# B&R Automation Studio project ProjectOrionBms
Automation Studio 4.12.6.106; technology packages: mapp 5.24.3, mappView 5.24.3

## Configuration Config1

CPU X90CP174.48-00, AutomationRuntime I4.93, Build 4.1.2, Safety 0.0, Vc V4.72.6

### Task classes (Cpu.sw)
```
Cyclic#1 (cycle 1000 us, tolerance 10000 us):
  INS <- INS.INS.prg
Cyclic#2 (cycle 4000 us, tolerance 20000 us):
  AMS_CAN <- AMS_and_Shunt.CAN.AMS_CAN.prg
  INV_CAN <- Inverters.CAN.CAN.prg
Cyclic#3 (cycle 10000 us, tolerance 20000 us):
  INV_CTRL <- Inverters.Control.Control.prg
Cyclic#4 (cycle 20000 us, tolerance 20000 us):
  INV_SM <- Inverters.Inv_statemachine.Inv_statemachine.prg
  SENSORS <- Sensors.Sensors.prg
  ACTUATORS <- Actuators.Output.prg
  DASHBOARD <- Dashboard.Dashboard.prg
  COOLING <- CoolingSystem.COOLING.prg
  file <- File.file.prg
  NewLogging <- Misc.DataLogging.NewLogging.prg
Cyclic#5 (cycle 50000 us, tolerance 50000 us):
  Simulation <- Inverters.Simulation.Simulation.prg [disabled]
  AMS_CTRL <- AMS_and_Shunt.AMS.prg
  SC <- SC.SafetyChain.prg
  SM <- SM.StateMachine.prg
  SENSOR_NET <- SensorNet.globalSensorNet.prg [disabled]
  ALARM_MAN <- Misc.AlarmManagement.AlarmManagement.prg
Cyclic#6 (cycle 100000 us, tolerance 100000 us):
  sampleST <- Misc.DataLogging.sampleST.prg [disabled]
  DATALOG <- Misc.DataLogging.DataLog.prg [disabled]
Binaries: TCData, udbdef, mvLoader, arsvcreg, ashwac, Role, ashwd, arconfig, sysconf, iomap, User, asfw, Config_1, Config, Config_2, Config_3, DataRecord, OpcUaMap, Acp10map, acp10cfg
Libraries: runtime, astime, standard, operator, AsIecCon, AsIODiag, brsystem, asstring, ArCan, brdkSIM, brdkUSB, AsIO, AsBrStr, sys_lib, FileIO, AsUSB, DataObj, brdkSTR, MpAlarmX, MpBase, MpData, NcGlobal, MpRecipe, sduVikings, MTTypes, dvframe, MTFilter, brdkFile, arssl, areventlog
```

### Hardware
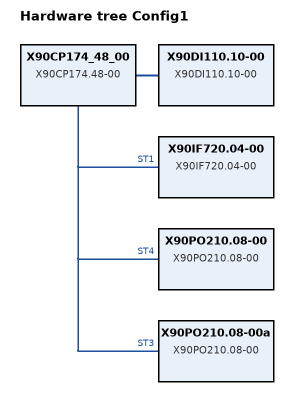
```
X90CP174_48_00 : X90CP174.48-00 v1.5.2.0  [X1 -> X1.SL]
  Module X1 (Type=X1, Virtual=true, Version=1.5.2.0)
    Connection (Connector=SL, TargetModule=X90CP174_48_00, TargetConnector=X1)
    ChannelConfig01 = 42
    DigitalFilterPin01 = 200
    ChannelConfig02 = 42
    DigitalFilterPin02 = 200
    ChannelConfig03 = 42
    DigitalFilterPin03 = 200
    ChannelConfig04 = 42
    DigitalFilterPin04 = 200
    ChannelConfig05 = 42
    DigitalFilterPin05 = 200
    ChannelConfig06 = 42
    DigitalFilterPin06 = 200
    ChannelConfig07 = 42
    DigitalFilterPin07 = 200
    ChannelConfig08 = 42
    DigitalFilterPin08 = 200
    ChannelConfig09 = 80
    ChannelConfig10 = 80
    ChannelConfig11 = 80
    ChannelConfig12 = 81
    ChannelConfig13 = 72
    DigitalFilterPin13 = 200
    ChannelConfig14 = 81
    ChannelConfig16 = 81
    ChannelConfig17 = 80
    ChannelConfig18 = 80
    ChannelConfig19 = 80
    ChannelConfig20 = 80
    ChannelConfig21 = 80
    ChannelConfig22 = 80
    ChannelConfig23 = 80
    IN2_InputFilter_Pin23 = 3
    ChannelConfig24 = 80
    ChannelConfig27 = 1
    ChannelConfig28 = 41
    DigitalFilterPin28 = 200
    ChannelConfig37 = 1
    LoadType37 = 2
    ChannelConfig38 = 1
    LoadType38 = 2
    ChannelConfig39 = 1
    ChannelConfig41 = 1
    LoadType41 = 2
    ChannelConfig42 = 1
    ChannelConfig45 = 1
    LoadType45 = 2
    ChannelConfig46 = 1
    LoadType46 = 2
    core = core1
  Connector IF2:
    ActivateDevice = 1
    Mode = Manual
    InternetAddress = 169.254.143.70
    SubnetMask = 255.255.0.0
    InaNodeNumber = 0
    ActivateSnmp = 2
  Connector IF3:
    DNAConfiguration = manual
    CycleTime = 1000
  ConfigurationID = Project_Config1
  UserPartitionSize = 100
  VolatileGlobalPvSize = 100000000
  IdleTaskClass = 5
  TaskClassIdleTime = 5000
  CyclicTaskClassCount = 6
  Cyclic1Duration = 1000
  Cyclic1Tolerance = 10000
  Cyclic2Duration = 4000
  Cyclic2Tolerance = 20000
  Cyclic3Duration = 10000
  Cyclic3Tolerance = 20000
  Cyclic4Duration = 20000
  Cyclic4Tolerance = 20000
  Cyclic5Duration = 50000
  Cyclic5Tolerance = 50000
  Cyclic6Duration = 100000
  Cyclic6Tolerance = 100000
  Cyclic7Duration = 100000
  Cyclic7Tolerance = 1000000
  Cyclic8Duration = 10000
  Cyclic8Tolerance = 30000000
  FileDevice1
  FileDeviceName1 = C
  FileDevicePath1 = C:/vikings/missions
  FileDevice2
  FileDeviceName2 = plc
  FileDevicePath2 = USER_PATH
  FtpUser1
  FtpUsername1 = viking  // viking
  FtpUserPassword1 = ZkV2vChQEXxJT0bhh2t/N5ZFPz9PChZjZfbJ7hc9Et0=  // viking
  FtpUserSalt1 = vdLLncGP
  FTPAccessRight1 = 0
  FTPdevice1 = ALL
  FtpUser2
  FtpUsername2 = usb  // usb
  FtpUserPassword2 = C1MDbg7H4C+9nkC1XVfE1m47HMH3DB0hBQDZaSBhzO4=  // usb
  FtpUserSalt2 = PgfniPeQ
  FTPAccessRight2 = 0
  FTPdevice2 = USB
  ActivateOpcUa = 1
  OpcUaInformationModels_PV_Version = 1
X90DI110.10-00 : X90DI110.10-00 v1.1.1.0  [ST -> X90CP174_48_00.ST2]
  Mode_DigIn01 = 22k_pnp
  InputFilter01 = 200
  Mode_DigIn02 = 22k_pnp
  InputFilter02 = 200
  Mode_DigIn03 = 22k_pnp
  InputFilter03 = 200
  Mode_DigIn04 = 22k_pnp
  Mode_DigIn05 = 22k_pnp
  Mode_DigIn06 = 22k_pnp
  Mode_DigIn07 = 22k_pnp
  InputFilter07 = 200
  Mode_DigIn08 = 22k_pnp
  Mode_DigIn09 = 22k_pnp
  InputFilter09 = 200
  Mode_DigIn10 = 22k_pnp
  InputFilter10 = 200
X90IF720.04-00 : X90IF720.04-00 v1.0.2.0  [ST -> X90CP174_48_00.ST1]
  Connector IF4:
    Baudrate = 115200
X90PO210.08-00 : X90PO210.08-00 v1.0.2.0  [ST -> X90CP174_48_00.ST4]
X90PO210.08-00a : X90PO210.08-00 v1.0.2.0  [ST -> X90CP174_48_00.ST3]
```

### IoMap.iom - X90CP174_48_00/IoMap.iom
```iecst
VAR_CONFIG
	::gCooling.outputs.do_fan[1] AT %QX."X1".DigitalOutput46;
	::gCooling.inputs.ai_coolingTemp[0] AT %IW."X1".AnalogInput17;
	::gCooling.inputs.ai_coolingTemp[1] AT %IW."X1".AnalogInput19;
	::gCooling.outputs.do_pump[1] AT %QX."X1".DigitalOutput45;
	::gCooling.outputs.do_fan[0] AT %QX."X1".DigitalOutput37;
	::gCooling.outputs.do_pump[0] AT %QX."X1".DigitalOutput38;
	::gSafetyChain.inputs.di_interlockWheelFR_OK AT %IX."X1".DigitalInput05;
	::gSafetyChain.inputs.di_shutdownRight_OK AT %IX."X1".DigitalInput07;
	::gSafetyChain.inputs.di_interlockWheelFL_OK AT %IX."X1".DigitalInput06;
	::gSafetyChain.inputs.di_interlockWheelRR_OK AT %IX."X1".DigitalInput08;
	::gSafetyChain.inputs.di_shutdownLeft_OK AT %IX."X1".DigitalInput01;
	::gSafetyChain.inputs.di_shutdownCockpit_OK AT %IX."X1".DigitalInput02;
	::gSafetyChain.inputs.di_inertiaSwitch_OK AT %IX."X1".DigitalInput03;
	::gSafetyChain.inputs.di_BOTS_OK AT %IX."X1".DigitalInput04;
	::gSafetyChain.inputs.di_TSMS_OK AT %IX."X1".DigitalInput13;
	::gSteeringAngle.inputs.angleSensor AT %IW."X1".AnalogInput20;
	::gTorqueSensor.inputs.torque2 AT %IW."X1".AnalogInput21;
	::gBraking.inputs.ai_brakePressureFront AT %IW."X1".AnalogInput22;
	::gTorqueSensor.inputs.torque1 AT %IW."X1".AnalogInput24;
	::gBraking.inputs.ai_brakePressureRear AT %IW."X1".AnalogInput18;
	::gInverters.inverter[0].inputs.di_deratingActive AT %IX."X90DI110.10-00".DigitalInput06;
	::gInverters.inverter[1].inputs.di_deratingActive AT %IX."X90DI110.10-00".DigitalInput04;
	::gInverters.inverter[2].inputs.di_deratingActive AT %IX."X90DI110.10-00".DigitalInput08;
	::gInverters.inverter[3].inputs.di_deratingActive AT %IX."X90DI110.10-00".DigitalInput05;
	::gInverters.inverter[0].outputs.do_enable AT %QX."X90PO210.08-00a".DigitalOutput01;
	::gInverters.inverter[1].outputs.do_enable AT %QX."X90PO210.08-00a".DigitalOutput07;
	::gInverters.inverter[3].outputs.do_enable AT %QX."X90PO210.08-00a".DigitalOutput06;
	::gInverters.inverter[2].outputs.do_torqueLimitActive AT %QX."X90PO210.08-00a".DigitalOutput02;
	::gInverters.inverter[0].outputs.do_torqueLimitActive AT %QX."X90PO210.08-00a".DigitalOutput03;
	::gInverters.inverter[1].outputs.do_torqueLimitActive AT %QX."X90PO210.08-00a".DigitalOutput08;
	::gInverters.output.do_enableInv34 AT %QX."X90PO210.08-00a".DigitalOutput04;
	::gInverters.inverter[2].outputs.do_enable AT %QX."X90PO210.08-00".DigitalOutput03;
	::gInverters.inverter[3].outputs.do_torqueLimitActive AT %QX."X90PO210.08-00".DigitalOutput02;
	::gInverters.output.do_enableInv12 AT %QX."X90PO210.08-00".DigitalOutput05;
	::gSafetyChain.inputs.di_TS_Container AT %IX."X90DI110.10-00".DigitalInput07;
	::gSafetyChain.inputs.di_interlockWheelRL_OK AT %IX."X90DI110.10-00".DigitalInput10;
	::gSafetyChain.inputs.di_supply AT %IX."X90DI110.10-00".DigitalInput09;
	::gSafetyChain.inputs.di_BSPD_OK AT %IX."X90DI110.10-00".DigitalInput03;
	::gSafetyChain.inputs.di_interlockHVD_OK AT %IX."X90DI110.10-00".DigitalInput01;
	::gSafetyChain.inputs.di_interlockTSMP_OK AT %IX."X90DI110.10-00".DigitalInput02;
	::gRTDS.outputs.do_RTDS AT %QX."X1".DigitalOutput41;
	::gBraking.outputs.do_brakeLight AT %QX."X1".DigitalOutput42;
	gRTDS.inputs.im_RTDS_Current AT %IW."X1".Current41;
	::gCooling.inputs.im_pumpCurrent[1] AT %IW."X1".Current45;
	::gCooling.inputs.im_pumpCurrent[0] AT %IW."X1".Current38;
	::gInverters.output.do_powerInv12 AT %QX."X1".DigitalOutput39;
	::gInverters.output.do_powerInv34 AT %QX."X1".DigitalOutput27;
	::gLowVoltageBattery.inputs.ai_voltage AT %IW."X1".AnalogInput12;
	::gLowVoltageBattery.inputs.ai_current AT %IW."X1".AnalogInput23;
	::gSafetyChain.inputs.di_interlockMotorRL_OK AT %IX."X1".DigitalInput28;
	::SENSORS:suspension.input.linearPosSensor[2] AT %IW."X1".AnalogInput16;
	::SENSORS:suspension.input.linearPosSensor[0] AT %IW."X1".AnalogInput14;
	::SENSORS:accelerometer.input.z_direction AT %IW."X1".AnalogInput09;
	::SENSORS:accelerometer.input.y_direction AT %IW."X1".AnalogInput10;
	::SENSORS:accelerometer.input.x_direction AT %IW."X1".AnalogInput11;
END_VAR
```

### Config_2.mpdatarecorder - X90CP174_48_00/mappServices/Config_2.mpdatarecorder
```
Element gDataRecorder (Type=mpdatarecorder)
  DataRecorder:
    MaxFileSize = 32000
    SaveInterval = 5000
```

### DataRecord.mpdatarecorder - X90CP174_48_00/mappServices/DataRecord.mpdatarecorder
```
Element gDataRecorderNew (Type=mpdatarecorder)
  DataRecorder:
    MaxNumberOfFiles = 4
    MaxFileSize = 32000
    DecimalDigits = 3
    SaveInterval = 2000
    FileNamePattern = Datalog_%H_%M_%S.csv
    TimeStampPattern = %H:%M:%S:%L
```

## Logical view

Binary libraries used (declarations not repeated): operator, runtime, astime, AsIecCon, standard, AsIODiag, brsystem, asstring, ArCan, brdkSIM, AsIO, AsBrStr, sys_lib, FileIO, AsUSB, DataObj, brdkSTR, NcGlobal, MTTypes 1.03.4, dvframe, MTFilter, MpAlarmX 5.24.3, MpBase, MpRecipe 5.24.3, MpData 5.24.3

- AS4_HW_X90PO210.08-00.exe (binary file, 1100199 bytes)
### Global.var - Global variables
```iecst
VAR
	gIsSimulation : BOOL;
END_VAR
```

### Package Logical/Libraries - Global libraries

### Library Logical/Libraries/brdkUSB (ANSIC, version 1.00.3)
Depends on: AsUSB, FileIO

#### brdkUSBConnect.c
```c
#include <bur/plctypes.h>
#include <string.h>
#ifdef __cplusplus
	extern "C"
	{
#endif

	#include "brdkUSB.h"

#ifdef __cplusplus
	};
#endif

#define true 1
#define false 0

/* Converts an UDINT into a STRING type */
static unsigned char brdkUSBuditoa(unsigned long Value, char* pString) {
	int i, j=0;
	pString[0] = 0;
	if (Value > 0) {
		while (Value > 0) {
			j++;
			for(i=j; i > 0 ; i--) {
				pString[i] =pString[i-1];
			}
			pString[0] = (Value % 10) + 48;			/* ASCII 48-57 = 0..9 */
			Value = (Value / 10);
		}
	}
	else {
		pString[0] = 48;								/* adds just a zero char  */
		pString[1] = 0;								/* ends the string  */
		j = 1;
	}
	return j;
}

void brdkUSBConnect(struct brdkUSBConnect* inst) {
	brdk_usb_connect_internal_typ* this = &inst->internal;
	int i,n,idx;
	char tmp[2];

	/* get list of all connected usb nodes */
	this->UsbNodeListGet_0.enable 					= true;
	this->UsbNodeListGet_0.pBuffer					= (UDINT)&this->nodeIdBuffer;
	this->UsbNodeListGet_0.bufferSize 				= sizeof(this->nodeIdBuffer);
	this->UsbNodeListGet_0.filterInterfaceClass 	= asusb_CLASS_MASS_STORAGE;
	this->UsbNodeListGet_0.filterInterfaceSubClass 	= 0;
	UsbNodeListGet(&this->UsbNodeListGet_0);
	if(this->UsbNodeListGet_0.status == ERR_OK || (this->UsbNodeListGet_0.status == asusbERR_USB_NOTFOUND && this->UsbNodeListGet_0.listNodes == 0)) {

		if(this->oldCnt != this->UsbNodeListGet_0.listNodes && this->UsbNodeListGet_0.listNodes > 0) {

			/* go through all list nodes and check if they have been added to the system */
			for (n = 0; n < this->UsbNodeListGet_0.listNodes; n++) {
				idx = -1;
				for (i = 0; i <= BRDK_USB_MAX_DEVICES; i++) {
					if (this->node[i].UsbNodeGet_0.nodeId == this->nodeIdBuffer[n]) {
						idx = this->nodeIdBuffer[n];
						break;
					}
				}
				if (idx == -1) {	/* device not found/added */
					for (i = 0; i <= BRDK_USB_MAX_DEVICES; i++) {
						if (this->node[i].UsbNodeGet_0.nodeId == 0) {
							this->node[i].UsbNodeGet_0.nodeId = this->nodeIdBuffer[n];
							break;
						}
					}
				}
			}
		}
		this->oldCnt = this->UsbNodeListGet_0.listNodes;
	}
	else if(inst->simulateMount && !this->simulationMountActivated) {
	/* find an avaible node index */
		for(i=0; i<= BRDK_USB_MAX_DEVICES; i++) {
			if(this->node[i].UsbNodeGet_0.nodeId == 0) {
				this->node[i].UsbNodeGet_0.nodeId = 4294967295LL;
				this->simulationMountActivated = true;
				break;
			}
		}
	}

	/* state machine for all usb nodes */
	for(i=0; i<= BRDK_USB_MAX_DEVICES; i++) {

		switch(this->node[i].state) {

			case 0: /* wait for id */
				if(this->node[i].UsbNodeGet_0.nodeId != 0) {
					this->node[i].UsbNodeGet_0.enable 		= (this->node[i].UsbNodeGet_0.nodeId < 4294967294LL);
					this->node[i].UsbNodeGet_0.pBuffer 		= (UDINT)&this->node[i].infoBuffer;
					this->node[i].UsbNodeGet_0.bufferSize 	= sizeof(usbNode_typ);
					UsbNodeGet(&this->node[i].UsbNodeGet_0);
					this->node[i].state 					= 10;
				}
				break;

			case 10:	/* get usb node info (interface name) */
				UsbNodeGet(&this->node[i].UsbNodeGet_0);
				switch(this->node[i].UsbNodeGet_0.status) {

					case ERR_OK:
						/* filter B&R technology guard from list */
						if(this->node[i].infoBuffer.vendorId == 1615 && this->node[i].infoBuffer.productId == 1001) this->node[i].state = 70;
						else {
							strcpy(this->node[i].device,"USB");
							brdkUSBuditoa(i,tmp);
							strcat(this->node[i].device,tmp);
							this->node[i].DevLink_0.pDevice = (UDINT)&this->node[i].device;
							strcpy(this->node[i].param, "/DEVICE=");
							strcat(this->node[i].param, this->node[i].infoBuffer.ifName);
							this->node[i].DevLink_0.pParam = (UDINT)&this->node[i].param;
							this->node[i].DevLink_0.enable = true;
							this->node[i].state = 20;
						}
						break;

					case asusbERR_USB_NOTFOUND:
						this->node[i].UsbNodeGet_0.nodeId = 0;
						memset(&this->node[i].infoBuffer,0,sizeof(usbNode_typ));
						this->node[i].state = 0;
						break;

					case ERR_FUB_ENABLE_FALSE:
						strcpy(this->node[i].device,"USB");
						brdkUSBuditoa(i,tmp);
						strcat(this->node[i].device,tmp);
						this->node[i].DevLink_0.pDevice = (UDINT)&this->node[i].device;
						strcpy(this->node[i].param, "/DEVICE=C:\\USB");
						this->node[i].DevLink_0.pParam = (UDINT)&this->node[i].param;
						this->node[i].DevLink_0.enable = true;
						this->node[i].state = 20;
						break;

				}
				break;

			case 20:	/* create device link */
				DevLink(&this->node[i].DevLink_0);
				switch(this->node[i].DevLink_0.status) {

					case ERR_OK:
						strcpy(inst->node[i].device,this->node[i].device);
						this->node[i].state = 40;
						break;

					case fiERR_DEVICE_ALREADY_EXIST:
						this->node[i].DevUnlink_0.enable 	= 1;
						this->node[i].DevUnlink_0.handle 	= this->node[i].DevLink_0.handle;
						this->node[i].state 				= 30;
						break;
				}
				break;

			case 30:	/* unlink device link */
				DevUnlink(&this->node[i].DevUnlink_0);
				switch(this->node[i].DevUnlink_0.status ) {

					case ERR_OK: case fiERR_DEVICE_INVALID_HANDLE:
						this->node[i].DevUnlink_0.enable 	= 0;
						DevUnlink(&this->node[i].DevUnlink_0);
						this->node[i].DevLink_0.enable 		= 0;
						DevLink(&this->node[i].DevLink_0);
						this->node[i].DevLink_0.enable 		= 1;
						this->node[i].devLinkFailCnt++;
						brdkUSBuditoa(this->node[i].devLinkFailCnt,tmp);
						strcat(this->node[i].device,tmp);
						this->node[i].DevLink_0.pDevice 	= (UDINT)&this->node[i].device;
						this->node[i].state					= 20;
						break;

				}
				break;

			case 40:	/* usb node ready - monitor node */
				UsbNodeGet(&this->node[i].UsbNodeGet_0);
				switch(this->node[i].UsbNodeGet_0.status) {

					case ERR_OK:
						if(inst->updateMemInfo || inst->node[i].totalMemory == 0) {
							this->node[i].DevMemInfo_0.enable = true;
							this->node[i].DevMemInfo_0.pDevice = this->node[i].DevLink_0.pDevice;
							this->node[i].state = 50;
						}
						break;

					case asusbERR_USB_NOTFOUND:
						strcpy(inst->node[i].device,"");
						this->node[i].DevUnlink_0.enable 	= true;
						this->node[i].DevUnlink_0.handle 	= this->node[i].DevLink_0.handle;
						this->node[i].state = 60;
						break;

					case ERR_FUB_ENABLE_FALSE:
						if(!inst->simulateMount && this->simulationMountActivated) {
							strcpy(inst->node[i].device,"");
							this->node[i].DevUnlink_0.enable 	= true;
							this->node[i].DevUnlink_0.handle 	= this->node[i].DevLink_0.handle;
							this->simulationMountActivated 		= false;
							this->node[i].state = 60;
						}
						break;

				}
				break;

			case 50:	/* read meminfo */
				DevMemInfo(&this->node[i].DevMemInfo_0);
				switch(this->node[i].DevMemInfo_0.status) {

					case ERR_OK:
						inst->node[i].freeMemory 	= this->node[i].DevMemInfo_0.freemem/1048576;	/* output must be in mb */
						inst->node[i].totalMemory 	= this->node[i].DevMemInfo_0.memsize/1048576;	/* output must be in mb */
						this->node[i].state 		= 40;
						break;

					case fiERR_DETMEMINFO: case fiERR_DEVICE_MANAGER:
						inst->node[i].freeMemory 	= -1;	/* output must be in mb */
						inst->node[i].totalMemory 	= -1;	/* output must be in mb */
						this->node[i].state 		= 40;
						break;

					case ERR_FUB_BUSY: break;
					default: this->node[i].state = 40; break;
				}
				break;

			case 60:	/* unlink device */
				DevUnlink(&this->node[i].DevUnlink_0);
				switch(this->node[i].DevUnlink_0.status ) {

					case ERR_OK: case fiERR_DEVICE_INVALID_HANDLE:
						this->node[i].DevUnlink_0.enable 	= false;
						DevUnlink(&this->node[i].DevUnlink_0);
						this->node[i].DevLink_0.enable 		= false;
						DevLink(&this->node[i].DevLink_0);
						this->node[i].UsbNodeGet_0.nodeId = 0;
						memset(&this->node[i].infoBuffer,0,sizeof(usbNode_typ));
						inst->node[i].freeMemory 	= 0;
						inst->node[i].totalMemory 	= 0;
						this->node[i].state = 0;
						break;

				}
				break;

			case 70:	/* B&R technology guard state */
				UsbNodeGet(&this->node[i].UsbNodeGet_0);
				switch(this->node[i].UsbNodeGet_0.status) {

					case ERR_OK: break;

					case asusbERR_USB_NOTFOUND:
						this->node[i].UsbNodeGet_0.nodeId = 0;
						memset(&this->node[i].infoBuffer,0,sizeof(usbNode_typ));
						this->node[i].state = 0;
						break;

				}
				break;

			case 1000:	/* simulate usb device */

				break;

		}
	}

	/* output status */
	for(i=0; i<= BRDK_USB_MAX_DEVICES; i++) {
		if(inst->node[i].device[0] != 0) {
			inst->status = BRDK_USB_STATUS_FB_READY;
			break;
		}
		else inst->status = BRDK_USB_STATUS_NO_USB_DEV_FOUND;
	}

	inst->updateMemInfo = 0;	/* reset update command */

}
```

### Library Logical/Libraries/sduVikings (IEC)

#### launchProfile.st
```iecst
FUNCTION_BLOCK launchProfile
	IF enable THEN

	ELSE
		FOR i := 0 TO 3 DO
			derating_output[i] := 1;
		END_FOR;
	END_IF;

END_FUNCTION_BLOCK
```

#### regenerativeBraking.st
```iecst
(* TODO: Add your comment here *)
FUNCTION_BLOCK regenerativeBraking
	IF NOT enable OR vehicle_lon_velocity < 5 OR torque_pedal > 0 THEN
		// Regenerative braking should be disabled if:
		//	 - Function block is not enabled
		// 	 - The vehicle velocity is below 5km/h
		//   - The torque pedal is pressed
		FOR i := 0 TO 3 DO
			negTrqLimSetpoint[i] := 0;
		END_FOR;
	ELSE
		// Regenerative braking is allowed
		IF brake_pressure = 0 THEN
			// Idle braking
			FOR i := 0 TO 3 DO
				negTrqLimSetpoint[i] := IDLE_MOTOR_TORQUE;
			END_FOR;
		ELSE
			// Control braking from brake pressure
			FOR i := 0 TO 3 DO
				// Calculate regen braking setpoint
				// Current algorithm is linear with the brake pressure offset by the idle motor torque
				// setpoint = idle_torque + gain * brake_pressure
				// The setpoint is then limited to within [0,1]
				negTrqLimSetpoint[i] := LIMIT(0, IDLE_MOTOR_TORQUE + REGEN_BRAKING_GAIN * brake_pressure, 1);
			END_FOR;
			// The setpoint can then be changed with the negative torque transfer from the TV algorithm
			// and limited to within [0,1]
			// Left, [0]&[2]
			negTrqLimSetpoint[0] := LIMIT(0, negTrqLimSetpoint[0] + negative_torque_transfer, 1);
			negTrqLimSetpoint[2] := LIMIT(0, negTrqLimSetpoint[2] + negative_torque_transfer, 1);
			// Right, [1]&[3]
			negTrqLimSetpoint[1] := LIMIT(0, negTrqLimSetpoint[1] - negative_torque_transfer, 1);
			negTrqLimSetpoint[3] := LIMIT(0, negTrqLimSetpoint[3] - negative_torque_transfer, 1);
		END_IF;
	END_IF;

	FOR i := 0 TO 3 DO
		negative_torque_limit[i] := 0;
		positive_torque_limit[i] := 1;
	END_FOR;
END_FUNCTION_BLOCK
```

#### torqueLimiter.st
```iecst
FUNCTION_BLOCK torqueLimiter

	IF enable THEN
		FOR i := 0 TO 3 DO
			derating_output[i] := max_torque/100.00;
		END_FOR;
	ELSE
		FOR i := 0 TO 3 DO
			derating_output[i] := 1;
		END_FOR;
	END_IF;

END_FUNCTION_BLOCK
```

#### tractionControl.st
```iecst
FUNCTION_BLOCK tractionControl
	IF enable THEN

	ELSE
		FOR i := 0 TO 3 DO
			derating_output[i] := 1;
		END_FOR;
	END_IF;

END_FUNCTION_BLOCK
```

### Library Logical/Libraries/brdkFile (ANSIC, version 2.00.0) - File handling library. Makes it easy to handle file devices and to do file handling.
Depends on: AsIODiag, AsUSB, FileIO, brdkSTR

#### brdkFile.typ - Data types
```iecst
TYPE
	brdk_file_dev_handler_int_typ : 	STRUCT  (*Internal variables.*)
		fileState : UINT; (*State of the file device handler.*)
		driveState : UINT; (*State of the drive handler.*)
		DevLink_0 : DevLink; (*Device link.*)
		DevUnlink_0 : DevUnlink; (*Device unlink.*)
		DirInfo_0 : DirInfo; (*Directory create.*)
		driveInternal : STRING[10]; (*Internal drive.*)
		drive : STRING[10]; (*Drive.*)
		deviceParam : STRING[BRDK_FILE_MAX_PATH_LEN]; (*Device parameter string.*)
		fileIdx : DINT; (*File index.*)
		activeHandles : ARRAY[0..BRDK_FILE_MAX_FILES_DEVICES_]OF UDINT; (*Active handles.*)
		internalRootHandle : UDINT; (*Internal drive.*)
		driveReady : BOOL; (*Drive ready to use.*)
		oldUseUSB : BOOL; (*Holds the old command.*)
		oldFileDeviceUseUSB : ARRAY[0..BRDK_FILE_MAX_FILES_DEVICES]OF BOOL; (*Holds the old command for each file device.*)
		usbOK : BOOL; (*USB drive present and ready to use.*)
		brdkFileCreateSubFolders_0 : brdkFileCreateSubFolders; (*Create sub folders.*)
		UsbNodeListGet_0 : UsbNodeListGet; (*Get list of USB nodes.*)
		UsbNodeGet_0 : UsbNodeGet; (*Get USB node.*)
		nodeId : ARRAY[0..BRDK_FILE_MAX_USB_NODES]OF UDINT; (*Node id buffer list.*)
		nodeIdx : USINT; (*Node id index.*)
		usbNode : usbNode_typ; (*Node info.*)
		oldUSBok : BOOL; (*Holds the old status.*)
		oldNodeId : UDINT; (*Holds the old node id.*)
		availableDeviceIndex : DINT; (*Last array index used in the available devices array*)
		availableUsbIndex : DINT; (*Last array index used in the available usb devices array*)
	END_STRUCT;
	brdk_file_dev_handler_sim_typ : 	STRUCT  (*Simulation options.*)
		pcRootFolder : STRING[BRDK_FILE_MAX_PATH_LEN] := 'plcRoot'; (*Path on the PC that will simulate the root of the controller. Default plcRoot -> C:\plcRoot\*)
		pcUSBDrive : brdk_file_drive_typ := D_DRIVE; (*Drive letter of the PC's USB. Default D:\.*)
		pcHDDrive : brdk_file_drive_typ := C_DRIVE; (*Drive letter of the PC's HD. Default C:\.*)
	END_STRUCT;
	brdk_file_dev_handler_setup_typ : 	STRUCT  (*Setup options.*)
		plcDrive : brdk_file_drive_typ := C_DRIVE; (*Drive letter of the controller flash. Default C:\.*)
		usbOverrule : BOOL := FALSE; (*Inserted USB stick will overrule internal flash if the USB stick is present.*)
		fileDevices : ARRAY[0..BRDK_FILE_MAX_FILES_DEVICES]OF brdk_file_file_devices_typ; (*File devices.*)
	END_STRUCT;
	brdk_file_drive_typ :
		( (*Drive selection. Default C:\.*)
		C_DRIVE := 0, (*C:\*)
		D_DRIVE := 1, (*D:\*)
		E_DRIVE := 2, (*E:\*)
		F_DRIVE := 3, (*F:\*)
		G_DRIVE := 4 (*G:\*)
		) := C_DRIVE;
	brdk_file_file_devices_typ : 	STRUCT  (*File devices setup.*)
		name : STRING[BRFK_FILE_MAX_FILE_DEVICE_LEN]; (*Name of the file device to be used as input for file functions.*)
		path : STRING[BRDK_FILE_MAX_PATH_LEN]; (*Folder path for the file device. Only the folders must be entered the drive is setup in the setup options. E.g. config.*)
		useUSB : BOOL := TRUE; (*Enable or disable that device can use a USB device. (True = Use USB if possible, False = Never use USB)*)
	END_STRUCT;
	brdk_file_create_subfold_int_typ : 	STRUCT  (*Internal variables.*)
		state : DINT; (*State of the function block.*)
		DirCreate_0 : DirCreate; (*Directory create.*)
		tmpPath : STRING[BRDK_FILE_MAX_PATH_LEN]; (*Temp path string.*)
		pathPos : DINT; (*Path position.*)
		tmpPathPos : DINT; (*Tmp path position.*)
		tmpLen : DINT; (*Temp length.*)
	END_STRUCT;
	brdk_file_read_internal_typ : 	STRUCT  (*Internal variables.*)
		state : DINT; (*State of the function block.*)
		FileOpen_0 : FileOpen; (*File open.*)
		FileClose_0 : FileClose; (*File close.*)
		FileRead_0 : FileRead; (*File read.*)
		offset : UDINT; (*Read offset.*)
	END_STRUCT;
	brdk_file_write_internal_typ : 	STRUCT  (*Internal variables.*)
		state : DINT; (*State of the function block.*)
		FileOpen_0 : FileOpen; (*File open.*)
		FileCreate_0 : FileCreate; (*File create.*)
		FileClose_0 : FileClose; (*File close.*)
		FileDelete_0 : FileDelete; (*File delete.*)
		FileWrite_0 : FileWrite; (*File write.*)
	END_STRUCT;
END_TYPE
```

#### brdkFile.var - Constants
```iecst
VAR CONSTANT
	BRDK_FILE_MAX_USB_NODES : USINT := 5; (*Maximum number of connected USB nodes. (5 means 6)*)
	BRDK_FILE_MAX_FILES_DEVICES_ : USINT := 10; (*Maximum numbers of file devices. (10 means 10)*)
	BRDK_FILE_MAX_FILES_DEVICES : USINT := 9; (*Maximum numbers of file devices. (9 means 10)*)
	BRDK_FILE_MAX_PATH_LEN : UINT := 200; (*Maximum length of a path.*)
	BRFK_FILE_MAX_FILE_DEVICE_LEN : UINT := 50; (*Maximum length of file device names.*)
END_VAR
```

#### brdkFile.fun - Functions and function blocks
```iecst
FUNCTION_BLOCK brdkFileDeviceHandler (*Easy file device handler. This function block makes file device handling easy. The idea of the function block is that you only need to create one file device name that can be used for both internal and usb flash.*) (*$GROUP=User,$CAT=User,$GROUPICON=User.png,$CATICON=User.png*)
	VAR_INPUT
		enable : BOOL := FALSE; (*Enables the function block.*)
		setup : brdk_file_dev_handler_setup_typ; (*Setup options.*)
		simulation : brdk_file_dev_handler_sim_typ; (*Simulation options.*)
		useUSB : BOOL := FALSE; (*Stores on the USB if it is possible. Can be auto selected in the setup options.*)
	END_VAR
	VAR_OUTPUT
		availableUSB : ARRAY[0..BRDK_FILE_MAX_FILES_DEVICES] OF STRING[BRFK_FILE_MAX_FILE_DEVICE_LEN]; (*List of available USB devices.*)
		availableDevices : ARRAY[0..BRDK_FILE_MAX_FILES_DEVICES] OF STRING[BRFK_FILE_MAX_FILE_DEVICE_LEN]; (*List of available PLC devices.*)
		ready : BOOL := FALSE; (*Means that all file devices have been created and are ready to use.*)
		description : STRING[200] := ''; (*Status description.*)
		status : UINT := 0; (*Status of FileIO function blocks.*)
	END_VAR
	VAR
		internal : brdk_file_dev_handler_int_typ; (*Internal variables.*)
	END_VAR
END_FUNCTION_BLOCK

FUNCTION_BLOCK brdkFileCreateSubFolders (*Creates folders based on a path string.*) (*$GROUP=User,$CAT=User,$GROUPICON=User.png,$CATICON=User.png*)
	VAR_INPUT
		enable : BOOL := FALSE; (*Enables the function block.*)
		path : STRING[BRDK_FILE_MAX_PATH_LEN] := ''; (*Path of folder to be created. Use \ to seperate folders.*)
		fileDevice : STRING[BRFK_FILE_MAX_FILE_DEVICE_LEN] := ''; (*File device name.*)
	END_VAR
	VAR_OUTPUT
		description : STRING[200] := ''; (*Status description.*)
		done : BOOL := FALSE; (*Function block done.*)
		status : UINT := 0; (*Status of DirCreate function block.*)
	END_VAR
	VAR
		internal : brdk_file_create_subfold_int_typ; (*Internal variables.*)
	END_VAR
END_FUNCTION_BLOCK

FUNCTION_BLOCK brdkFileWrite (*Write data to a file.*) (*$GROUP=User,$CAT=User,$GROUPICON=User.png,$CATICON=User.png*)
	VAR_INPUT
		enable : BOOL := FALSE; (*Enables the function block.*)
		pFileDevice : UDINT := 0; (*String pointer to file device.*)
		pFileName : UDINT := 0; (*String pointer to file name.If the file does not exist it will be created.*)
		pData : UDINT := 0; (*Pointer to the data that must be written to the file.*)
		dataLength : UDINT := 0; (*Length of the data that must be written. If 0 is specified \0 will end the data.*)
		overwrite : BOOL := FALSE; (*Overwrite existing file. If not set the data will be appended to existing file.*)
	END_VAR
	VAR_OUTPUT
		status : UINT := 0; (*Status of the function block.*)
	END_VAR
	VAR
		internal : brdk_file_write_internal_typ; (*Internal variables.*)
	END_VAR
END_FUNCTION_BLOCK

FUNCTION_BLOCK brdkFileRead (*Read data from a file.*) (*$GROUP=User,$CAT=User,$GROUPICON=User.png,$CATICON=User.png*)
	VAR_INPUT
		enable : BOOL := FALSE; (*Enables the function block.*)
		pFileDevice : UDINT := 0; (*String pointer to file device.*)
		pFileName : UDINT := 0; (*String pointer to file name.*)
		pData : UDINT := 0; (*Pointer to the data where the data is read to.*)
		dataLength : UDINT := 0; (*Length of the read data buffer.*)
	END_VAR
	VAR_OUTPUT
		status : UINT := 0; (*Status of the function block.*)
		readLength : UDINT := 0; (*Length of the read data.*)
	END_VAR
	VAR
		internal : brdk_file_read_internal_typ; (*Internal variables.*)
	END_VAR
END_FUNCTION_BLOCK
```

#### brdkFileDeviceHandler.c - Easy file device handler.
```c
#include <brdkFile_func.h>

#define BR_TG_VENDOR_ID 1615
#define BR_TG_PRODUCT_ID 1001

void brdkFileDeviceHandler(struct brdkFileDeviceHandler* inst) {
	brdk_file_dev_handler_int_typ* this 	= (brdk_file_dev_handler_int_typ*)&inst->internal;		/* pointer to the internal structure */
	brdk_file_dev_handler_setup_typ* setup 	= (brdk_file_dev_handler_setup_typ*)&inst->setup;		/* pointer to the setup structure */
	brdk_file_dev_handler_sim_typ* sim 		= (brdk_file_dev_handler_sim_typ*)&inst->simulation;	/* pointer to the simulation structure */
	char tmpStr[200];

	if(inst->enable) {

		/* check whether the controller is beeing simulated and watch the usb status */
		if(!DiagCpuIsSimulated()) {
			if(!this->UsbNodeGet_0.enable) this->UsbNodeListGet_0.enable = true;
			this->UsbNodeListGet_0.pBuffer					= (unsigned long)&this->nodeId;
			this->UsbNodeListGet_0.bufferSize 				= sizeof(this->nodeId);
			this->UsbNodeListGet_0.filterInterfaceClass 	= asusb_CLASS_MASS_STORAGE;
			this->UsbNodeListGet_0.filterInterfaceSubClass 	= asusb_SUBCLASS_SCSI_COMMAND_SET;
			UsbNodeListGet(&this->UsbNodeListGet_0);
			if(this->UsbNodeListGet_0.status == asusbERR_USB_NOTFOUND) {
				this->nodeIdx 	= 0;
				this->usbOK 	= false;
			}

			this->UsbNodeGet_0.enable 		= true;
			this->UsbNodeGet_0.nodeId 		= this->nodeId[this->nodeIdx];
			this->UsbNodeGet_0.pBuffer 		= (unsigned long)&this->usbNode;
			this->UsbNodeGet_0.bufferSize 	= sizeof(this->usbNode);
			UsbNodeGet(&this->UsbNodeGet_0);
			if(this->UsbNodeGet_0.status == ERR_OK) {
				if(this->usbNode.vendorId == BR_TG_VENDOR_ID && this->usbNode.productId == BR_TG_PRODUCT_ID) {
					this->UsbNodeGet_0.enable = false;
					UsbNodeGet(&this->UsbNodeGet_0);
					this->nodeIdx++;
				}
				else this->usbOK = true;
			}
			else if(this->UsbNodeGet_0.status == asusbERR_USB_NOTFOUND) {
				this->UsbNodeListGet_0.enable = true;
				this->nodeIdx = 0;
				this->usbOK = false;
			}
			if(this->oldNodeId != this->UsbNodeGet_0.nodeId) this->usbOK = false;
			this->oldNodeId = this->UsbNodeGet_0.nodeId;
		}
		else {
			/* look for USB root folder */
			if(this->DirInfo_0.pDevice != 0) {
				this->DirInfo_0.enable 	= true;
				this->DirInfo_0.pPath 	= (unsigned long)"";
				DirInfo(&this->DirInfo_0);
				switch(this->DirInfo_0.status) {
					case 0: this->usbOK = true; break;
					case 20723: this->usbOK = false; break;
					default: break;
				}
			}
		}
		if(setup->usbOverrule) inst->useUSB = this->usbOK;	/* USB stick will overrule */
	}
	else {
		this->usbOK 					= false;
		this->nodeIdx 					= 0;
		this->DirInfo_0.enable 			= false;
		DirInfo(&this->DirInfo_0);
		this->UsbNodeGet_0.enable 		= false;
		UsbNodeGet(&this->UsbNodeGet_0);
		this->UsbNodeListGet_0.enable 	= false;
		UsbNodeListGet(&this->UsbNodeListGet_0);
	}

	/* drive handler */
	switch(this->driveState) {

		case 0:
			if(inst->enable) {
				if(!DiagCpuIsSimulated()) {										// If the plc is not simulated
					if((inst->useUSB && this->usbOK) || !inst->useUSB) {
						this->driveReady = true;
						if(!inst->useUSB)getDrive(setup->plcDrive,this->drive);
						else brdkStrCpy((unsigned long)this->drive,(unsigned long)this->usbNode.ifName);
						getDrive(setup->plcDrive,this->driveInternal);
						this->driveState = 499;
					}
				}
				else {															// If the plc is simulated
					this->DevLink_0.enable 	= true;
					this->DevLink_0.pDevice = (unsigned long)"INTUSB";
					this->DevLink_0.pParam 	= buildParameterString(getDrive(sim->pcUSBDrive,this->drive),(char*)&"",(char*)&this->deviceParam);
					brdkStrCpy((unsigned long)this->driveInternal, (unsigned long) this->drive);
					this->driveState 		= 100;
				}
			}
			break;

		case 100:	/* create a file device for finding an attached usb flash */
			DevLink(&this->DevLink_0);
			if(this->DevLink_0.status != ERR_FUB_BUSY) {
				if(this->DevLink_0.status == ERR_OK || this->DevLink_0.status == fiERR_DEVICE_ALREADY_EXIST) {
					this->DirInfo_0.pDevice = this->DevLink_0.pDevice;
					this->DevLink_0.enable 	= false;
					DevLink(&this->DevLink_0);
					this->driveState 		= 110;
				}
				else {
					inst->status = this->DevLink_0.status;
					this->DevLink_0.enable 	= false;
					DevLink(&this->DevLink_0);
					brdkStrCpy((unsigned long)inst->description,(unsigned long)"error calling DevLink. Flip enable to reset fb.");
					this->driveState = 900;
				}
			}
			break;

		case 110:	/* wait for DirInfo to have been call once. Fb is call above */
			switch(this->DirInfo_0.status) {

				case 0: case 20723:
					if(!inst->useUSB) {
						getDrive(sim->pcHDDrive,this->drive);
						brdkStrCat((unsigned long)this->drive,(unsigned long)sim->pcRootFolder);
					}
					else getDrive(sim->pcUSBDrive,this->drive);
					getDrive(sim->pcHDDrive,this->driveInternal);
					brdkStrCat((unsigned long)this->driveInternal,(unsigned long)sim->pcRootFolder);

					this->driveState = 499;
					this->driveReady = true;
					break;

				case 65534: case 65535: break;

				default:
					inst->status 			= this->DirInfo_0.status;
					this->DirInfo_0.enable 	= false;
					DirInfo(&this->DirInfo_0);
					brdkStrCpy((unsigned long)inst->description,(unsigned long)"error calling DirInfo. Flip enable to reset fb.");
					this->driveReady = false;
					this->driveState = 900;
					break;
			}
			break;

		case 499:	/* waiting for file devices to be ready */
			if(!inst->enable) {
				this->driveReady = false;
				this->driveState = 900;
			}
			else if(inst->ready) this->driveState = 500;
			break;

		case 500:	/* check if USB status changes */
			if(!inst->enable) {
				this->driveReady = false;
				this->driveState = 900;
			}
			else if((this->oldUseUSB != inst->useUSB) || (inst->useUSB && (this->oldUSBok != this->usbOK))) {	/* usb must be used and the ok status has changed */
				this->driveReady = false;
				if(inst->useUSB && !this->usbOK) brdkStrCpy((unsigned long)inst->description,(unsigned long)"USB not ready. Turn off useUSB command.");
				else this->driveState = 510;
			}
			this->oldUseUSB = inst->useUSB;
			this->oldUSBok 	= this->usbOK;
			this->oldNodeId = this->UsbNodeGet_0.nodeId;
			break;

		case 510:	/* select the new drive */
			if(!DiagCpuIsSimulated()) {																// check if the controller is simulated
				if(!inst->useUSB)getDrive(setup->plcDrive,this->drive);
				else brdkStrCpy((unsigned long)this->drive,(unsigned long)this->usbNode.ifName);	// If useUSB set drive to new usb
				getDrive(setup->plcDrive,this->driveInternal);
			}
			else {
				if(!inst->useUSB) {
					getDrive(sim->pcHDDrive,this->drive);											// Get internal drive
					brdkStrCat((unsigned long)this->drive,(unsigned long)sim->pcRootFolder);		// Add folder name
				}
				else getDrive(sim->pcUSBDrive,this->drive);											// If useUSB and its a simulated PLC set drive to pcUSBDrive
				getDrive(sim->pcHDDrive,this->driveInternal);											// Get internal drive
				brdkStrCat((unsigned long)this->driveInternal,(unsigned long)sim->pcRootFolder);		// Add folder name
			}
			this->driveReady = true;
			this->driveState = 499;
			break;

		case 900:	/* error state */
			this->driveReady = false;
			if(!inst->enable) {
				inst->status 		= 0;
				this->driveState 	= 0;
			}
			break;

	}

	/* file device handler */
	switch(this->fileState) {

		case 0: /* wait for a drive */
			if(inst->enable) {
				if(this->driveReady) {
					this->DevLink_0.enable 	= true;
					this->DevLink_0.pDevice = (unsigned long)"ROOT";
					this->DevLink_0.pParam 	= buildParameterString((char*)&this->drive,(char*)&"",(char*)&this->deviceParam);
					brdkStrCpy((unsigned long)inst->description,(unsigned long)"creates a devlink for the drive root");
					this->fileState 		= 10;
				}
			}
			else {
				inst->ready = false;
			}
			break;

		case 10: /* Create drive for root */
			DevLink(&this->DevLink_0);
			if(this->DevLink_0.status != ERR_FUB_BUSY) {
				if(this->DevLink_0.status == ERR_OK) {
					brdkStrCpy((unsigned long)inst->availableDevices[0],this->DevLink_0.pDevice);
					this->activeHandles[0] = this->DevLink_0.handle;
					this->DevLink_0.enable 	= false;
					DevLink(&this->DevLink_0);
					this->fileIdx = 0;
					if(setup->fileDevices[this->fileIdx].name[0] != 0) {
						if(!this->usbOK || (this->usbOK && setup->fileDevices[this->fileIdx].useUSB && inst->useUSB)) this->brdkFileCreateSubFolders_0.enable = true;
						else this->brdkFileCreateSubFolders_0.enable = false;
						brdkStrCpy((unsigned long)this->brdkFileCreateSubFolders_0.path,(unsigned long)setup->fileDevices[this->fileIdx].path);
						brdkStrCpy((unsigned long)this->brdkFileCreateSubFolders_0.fileDevice,this->DevLink_0.pDevice);
						brdkFileCreateSubFolders(&this->brdkFileCreateSubFolders_0);
						brdkStrCpy((unsigned long)inst->description,(unsigned long)"creates the needed folders");
						this->fileState = 20;
					}
					else this->fileState = 80;
				}
				else if(this->DevLink_0.status == fiERR_DEVICE_ALREADY_EXIST) {
					if(this->DevLink_0.handle != 0) {
						inst->status = this->DevLink_0.status;
						this->DevLink_0.enable 	= false;
						DevLink(&this->DevLink_0);
						brdkStrCpy((unsigned long)inst->description,(unsigned long)"Device ");
						brdkStrCat((unsigned long)inst->description,this->DevLink_0.pDevice);
						brdkStrCat((unsigned long)inst->description,(unsigned long)" already exists. Reboot controller to kill the old device.");
						this->fileState = 900;
					}
					else {
						this->DevUnlink_0.enable = true;
						this->DevUnlink_0.handle = this->DevLink_0.handle;
						this->DevLink_0.enable 	= false;
						DevLink(&this->DevLink_0);
						this->fileState = 60;
					}
				}
				else {
					brdkStrCpy((unsigned long)inst->description,(unsigned long)"error calling DevLink. Flip enable to reset fb.");
					inst->status 			= this->DevLink_0.status;
					this->DevLink_0.enable 	= false;
					DevLink(&this->DevLink_0);
					this->fileState 		= 900;
				}
			}
			break;

		case 20: /* Create the needed folders */
			brdkFileCreateSubFolders(&this->brdkFileCreateSubFolders_0);
			if(this->brdkFileCreateSubFolders_0.done || !this->brdkFileCreateSubFolders_0.enable) {
				this->brdkFileCreateSubFolders_0.enable = false;
				brdkFileCreateSubFolders(&this->brdkFileCreateSubFolders_0);
				this->fileIdx++;
				if(setup->fileDevices[this->fileIdx].name[0] != 0 && setup->fileDevices[this->fileIdx].path[0] != 0) {
					if(!this->usbOK || (this->usbOK && setup->fileDevices[this->fileIdx].useUSB && inst->useUSB)){
						this->brdkFileCreateSubFolders_0.enable = true;
						brdkStrCpy((unsigned long)this->brdkFileCreateSubFolders_0.path,(unsigned long)setup->fileDevices[this->fileIdx].path);
						brdkFileCreateSubFolders(&this->brdkFileCreateSubFolders_0);
					}
				}
				else {
					if(this->usbOK){
						// USB device present => Create folders and device internally
						this->fileIdx = 0;
						this->DevLink_0.enable 	= true;
						this->DevLink_0.pDevice = (unsigned long)"INTERNAL_ROOT";
						this->DevLink_0.pParam 	= buildParameterString((char*)&this->driveInternal,(char*)&"",(char*)&this->deviceParam);
						brdkStrCpy((unsigned long)inst->description,(unsigned long)"creates a devlink for the drive internal");
						this->fileState = 30;
					}else{
						// No USB device present =>  Change device to ROOT device (internally)
						this->internalRootHandle = this->activeHandles[0];
						this->fileIdx = 0;
						this->DevLink_0.enable 	= true;
						this->DevLink_0.pDevice = (unsigned long)setup->fileDevices[this->fileIdx].name;
						this->DevLink_0.pParam 	= buildParameterString((char*)&this->drive,(char*)&setup->fileDevices[this->fileIdx].path,(char*)&this->deviceParam);
						this->fileState = 50;
					}
				}
			}

			else if(this->brdkFileCreateSubFolders_0.status == fiERR_FILE_DEVICE) {
				if(DiagCpuIsSimulated()) {
					this->DevUnlink_0.enable 	= true;
					this->DevUnlink_0.handle 	= this->activeHandles[0];
					this->activeHandles[0] 		= 0;
					DevUnlink(&this->DevUnlink_0);
					this->brdkFileCreateSubFolders_0.enable = false;
					brdkFileCreateSubFolders(&this->brdkFileCreateSubFolders_0);
					this->fileState 			= 200;
				}
				else {
					brdkStrCpy((unsigned long)inst->description,(unsigned long)"error calling brdkFileCreateSubFolders. Flip enable to reset fb.");
					inst->status 				= this->brdkFileCreateSubFolders_0.status;
					this->brdkFileCreateSubFolders_0.enable = false;
					brdkFileCreateSubFolders(&this->brdkFileCreateSubFolders_0);
					this->fileState 			= 900;
				}
			}
			else if(this->brdkFileCreateSubFolders_0.status != ERR_FUB_BUSY) brdkStrCpy((unsigned long)inst->description,(unsigned long)"error calling brdkFileCreateSubFolders. Check fb for error codes.");

			break;

		case 30: /* Create devices internally */
			DevLink(&this->DevLink_0);
			if(this->DevLink_0.status != ERR_FUB_BUSY) {
				if(this->DevLink_0.status == ERR_OK) {
					this->internalRootHandle = this->DevLink_0.handle;
					this->DevLink_0.enable 	= false;
					DevLink(&this->DevLink_0);
					brdkStrCpy((unsigned long)this->brdkFileCreateSubFolders_0.path,(unsigned long)setup->fileDevices[this->fileIdx].path);
					brdkStrCpy((unsigned long)this->brdkFileCreateSubFolders_0.fileDevice,this->DevLink_0.pDevice);
					this->brdkFileCreateSubFolders_0.enable = true;
					brdkFileCreateSubFolders(&this->brdkFileCreateSubFolders_0);
					brdkStrCpy((unsigned long)inst->description,(unsigned long)"creates the needed folders internally");
					this->fileState = 40;
				}
				else if(this->DevLink_0.status == fiERR_DEVICE_ALREADY_EXIST) {
					if(this->DevLink_0.handle != 0) {
						inst->status = this->DevLink_0.status;
						this->DevLink_0.enable 	= false;
						DevLink(&this->DevLink_0);
						brdkStrCpy((unsigned long)inst->description,(unsigned long)"Device ");
						brdkStrCat((unsigned long)inst->description,this->DevLink_0.pDevice);
						brdkStrCat((unsigned long)inst->description,(unsigned long)" already exists. Reboot controller to kill the old device.");
						this->fileState = 900;
					}
					else {
						this->DevUnlink_0.enable = true;
						this->DevUnlink_0.handle = this->DevLink_0.handle;
						this->DevLink_0.enable 	= false;
						DevLink(&this->DevLink_0);
						this->fileState = 70;
					}
				}
				else {
					brdkStrCpy((unsigned long)inst->description,(unsigned long)"error calling DevLink. Flip enable to reset fb.");
					inst->status 			= this->DevLink_0.status;
					this->DevLink_0.enable 	= false;
					DevLink(&this->DevLink_0);
					this->fileState 		= 900;
				}
			}
			break;

		case 40: /* Create folders internally */
			brdkFileCreateSubFolders(&this->brdkFileCreateSubFolders_0);
			if(this->brdkFileCreateSubFolders_0.done || !this->brdkFileCreateSubFolders_0.enable) {
				this->brdkFileCreateSubFolders_0.enable = false;
				brdkFileCreateSubFolders(&this->brdkFileCreateSubFolders_0);
				this->fileIdx++;
				if(setup->fileDevices[this->fileIdx].name[0] != 0 && setup->fileDevices[this->fileIdx].path[0] != 0) {
					if(!setup->fileDevices[this->fileIdx].useUSB && inst->useUSB){
						this->brdkFileCreateSubFolders_0.enable = true;
						brdkStrCpy((unsigned long)this->brdkFileCreateSubFolders_0.path,(unsigned long)setup->fileDevices[this->fileIdx].path);
						brdkFileCreateSubFolders(&this->brdkFileCreateSubFolders_0);
					}
				}
				else {
					this->fileIdx = 0;
					this->DevLink_0.enable 	= true;
					this->DevLink_0.pDevice = (unsigned long)setup->fileDevices[this->fileIdx].name;
					this->DevLink_0.pParam 	= buildParameterString((char*)&this->drive,(char*)&setup->fileDevices[this->fileIdx].path,(char*)&this->deviceParam);
					brdkStrCpy((unsigned long)inst->description,(unsigned long)"creates the needed file devices");
					this->fileState = 50;
				}
			}

			else if(this->brdkFileCreateSubFolders_0.status == fiERR_FILE_DEVICE) {
				if(DiagCpuIsSimulated()) {
					this->DevUnlink_0.enable 	= true;
					this->DevUnlink_0.handle 	= this->activeHandles[0];
					this->activeHandles[0] 		= 0;
					DevUnlink(&this->DevUnlink_0);
					this->brdkFileCreateSubFolders_0.enable = false;
					brdkFileCreateSubFolders(&this->brdkFileCreateSubFolders_0);
					this->fileState 			= 200;
				}
				else {
					brdkStrCpy((unsigned long)inst->description,(unsigned long)"error calling brdkFileCreateSubFolders. Flip enable to reset fb.");
					inst->status 				= this->brdkFileCreateSubFolders_0.status;
					this->brdkFileCreateSubFolders_0.enable = false;
					brdkFileCreateSubFolders(&this->brdkFileCreateSubFolders_0);
					this->fileState 			= 900;
				}
			}
			else if(this->brdkFileCreateSubFolders_0.status != ERR_FUB_BUSY) brdkStrCpy((unsigned long)inst->description,(unsigned long)"error calling brdkFileCreateSubFolders. Check fb for error codes.");

			break;

		case 50: /* Create USB devices */
			DevLink(&this->DevLink_0);
			if(this->DevLink_0.status != ERR_FUB_BUSY) {
				if(this->DevLink_0.status == ERR_OK) {
					this->activeHandles[this->fileIdx+1] = this->DevLink_0.handle;
					this->DevLink_0.enable 	= false;
					DevLink(&this->DevLink_0);
					this->fileIdx++;
					if(setup->fileDevices[this->fileIdx].name[0] != 0 && setup->fileDevices[this->fileIdx].path[0] != 0) {
						this->DevLink_0.enable 	= true;
						this->DevLink_0.pDevice = (unsigned long)setup->fileDevices[this->fileIdx].name;
						if(setup->fileDevices[this->fileIdx].useUSB) this->DevLink_0.pParam 	= buildParameterString((char*)&this->drive,(char*)&setup->fileDevices[this->fileIdx].path,(char*)&this->deviceParam);
						else{
							if(!DiagCpuIsSimulated()) getDrive(setup->plcDrive,this->driveInternal);
							else {
								getDrive(sim->pcHDDrive,this->driveInternal);
								brdkStrCat((unsigned long)this->driveInternal,(unsigned long)sim->pcRootFolder);
							}
							this->DevLink_0.pParam 	= buildParameterString((char*)&this->driveInternal,(char*)&setup->fileDevices[this->fileIdx].path,(char*)&this->deviceParam);
						}
					}
					else {
						inst->ready = true;
						brdkStrCpy((unsigned long)inst->description,(unsigned long)"all file devices are ready to use");
						this->fileState = 80;
					}
				}
				else {
					brdkStrCpy((unsigned long)inst->description,(unsigned long)"error calling DevLink. Flip enable to reset fb.");
					inst->status 			= this->DevLink_0.status;
					this->DevLink_0.enable 	= false;
					DevLink(&this->DevLink_0);
					this->fileState 		= 900;
				}
			}
			this->oldFileDeviceUseUSB[this->fileIdx] = setup->fileDevices[this->fileIdx].useUSB;
			break;

		case 60: /* Unlink root device */
			DevUnlink(&this->DevUnlink_0);
			if(this->DevUnlink_0.status != ERR_FUB_BUSY) {
				if(this->DevUnlink_0.status == ERR_OK) {
					this->DevUnlink_0.enable = false;
					DevUnlink(&this->DevUnlink_0);
					this->DevLink_0.enable 	= true;
					this->DevLink_0.pDevice = (unsigned long)"ROOT";
					this->DevLink_0.pParam 	= buildParameterString((char*)&this->drive,(char*)&"",(char*)&this->deviceParam);
					this->fileState 		= 10;
				}
				else {
					brdkStrCpy((unsigned long)inst->description,(unsigned long)"error calling DevUnlink. Flip enable to reset fb.");
					inst->status 				= this->DevUnlink_0.status;
					this->DevUnlink_0.enable 	= false;
					DevUnlink(&this->DevUnlink_0);
					this->fileState 			= 900;
				}
			}
			break;

		case 70: /* Unlink root device */
			DevUnlink(&this->DevUnlink_0);
			if(this->DevUnlink_0.status != ERR_FUB_BUSY) {
				if(this->DevUnlink_0.status == ERR_OK) {
					this->DevUnlink_0.enable = false;
					DevUnlink(&this->DevUnlink_0);
					this->DevLink_0.enable 	= true;
					this->DevLink_0.pDevice = (unsigned long)"ROOT";
					this->DevLink_0.pParam 	= buildParameterString((char*)&this->drive,(char*)&"",(char*)&this->deviceParam);
					this->fileState 		= 30;
				}
				else {
					brdkStrCpy((unsigned long)inst->description,(unsigned long)"error calling DevUnlink. Flip enable to reset fb.");
					inst->status 				= this->DevUnlink_0.status;
					this->DevUnlink_0.enable 	= false;
					DevUnlink(&this->DevUnlink_0);
					this->fileState 			= 900;
				}
			}
			break;

		case 80: /* Prepare for available list t be created */
			this->fileIdx 				= 0;
			this->availableDeviceIndex 	= 0;
			this->availableUsbIndex	 	= 0;
			this->fileState 			= 90;
			break;

		case 90: /* Create the available lists */
			brdkStrCpy((unsigned long)inst->availableDevices[this->fileIdx],(unsigned long)"");
			brdkStrCpy((unsigned long)inst->availableUSB[this->fileIdx]	   ,(unsigned long)"");
			if(this->fileIdx != 0){
				if(brdkStrCmp((unsigned long)setup->fileDevices[this->fileIdx-1].name,(unsigned long)"") != 0){
					if(setup->fileDevices[this->fileIdx-1].useUSB && inst->useUSB && this->usbOK ){
						brdkStrCpy((unsigned long)inst->availableUSB[this->availableUsbIndex],(unsigned long)setup->fileDevices[this->fileIdx-1].name);
						this->availableUsbIndex++;
					}
					else{
						brdkStrCpy((unsigned long)inst->availableDevices[this->availableDeviceIndex],(unsigned long)setup->fileDevices[this->fileIdx-1].name);
						this->availableDeviceIndex++;
					}
				}
			}
			else{
				if(inst->useUSB && this->usbOK){
					brdkStrCpy((unsigned long)inst->availableUSB[this->fileIdx],(unsigned long)"ROOT");
					this->availableUsbIndex++;
					brdkStrCpy((unsigned long)inst->availableDevices[this->fileIdx],(unsigned long)"INTERNAL_ROOT");
					this->availableDeviceIndex++;
				}
				else{
					brdkStrCpy((unsigned long)inst->availableDevices[this->fileIdx],(unsigned long)"ROOT");
					this->availableDeviceIndex++;
				}
			}
			this->fileIdx++;
			if(this->fileIdx >= BRDK_FILE_MAX_FILES_DEVICES){
				this->fileState 		= 100;
			}
			break;

		case 100:
			if(!inst->enable) {
				inst->ready 	= false;
				this->fileState = 900;
			}

			if(this->fileIdx < BRDK_FILE_MAX_FILES_DEVICES) {
				this->fileIdx++;
			}
			else {
				this->fileIdx = 0;
			}

			if(!(this->oldFileDeviceUseUSB[this->fileIdx] == setup->fileDevices[this->fileIdx].useUSB) && this->activeHandles[this->fileIdx+1] != 0 && this->usbOK){
				inst->ready 				= false;
				this->DevUnlink_0.enable 	= true;
				this->DevUnlink_0.handle 	= this->activeHandles[this->fileIdx+1];
				DevUnlink(&this->DevUnlink_0);
				brdkStrCpy((unsigned long)inst->description,(unsigned long)"removing device.");
				this->fileState 			= 300;
			}
			this->oldFileDeviceUseUSB[this->fileIdx] = setup->fileDevices[this->fileIdx].useUSB;

			if(!this->driveReady) {
				inst->ready = false;
				if(this->activeHandles[0] != 0) {
					this->fileIdx 				= 0;
					this->DevUnlink_0.enable 	= true;
					this->DevUnlink_0.handle 	= this->activeHandles[this->fileIdx];
					this->fileState 			= 110;
				}
				else this->fileState = 0;
			}

		break;

		case 110:	/* unlink file devices */
			DevUnlink(&this->DevUnlink_0);
			if(this->DevUnlink_0.status != ERR_FUB_BUSY) {
				if(this->DevUnlink_0.status == ERR_OK) {
					this->activeHandles[this->fileIdx] = 0;
					this->fileIdx++;
					this->DevUnlink_0.enable = false;
					DevUnlink(&this->DevUnlink_0);
					if(this->activeHandles[this->fileIdx] != 0) {
						this->DevUnlink_0.enable = true;
						this->DevUnlink_0.handle = this->activeHandles[this->fileIdx];
					}
					else this->fileState = 0;
				}
				else {
					brdkStrCpy((unsigned long)inst->description,(unsigned long)"error calling DevUnlink. Flip enable to reset fb.");
					inst->status 				= this->DevUnlink_0.status;
					this->DevUnlink_0.enable 	= false;
					DevUnlink(&this->DevUnlink_0);
					this->fileState 			= 900;
				}
			}
			break;

		case 200:
			DevUnlink(&this->DevUnlink_0);
			if(this->DevUnlink_0.status != ERR_FUB_BUSY) {
				if(this->DevUnlink_0.status == ERR_OK) {
					this->DevUnlink_0.enable = false;
					DevUnlink(&this->DevUnlink_0);
					this->DevLink_0.enable 	= true;
					this->DevLink_0.pDevice = (unsigned long)"tmpRoot";
					this->DevLink_0.pParam 	= buildParameterString(getDrive(sim->pcHDDrive,tmpStr),(char*)&"",(char*)&this->deviceParam);
					brdkStrCpy((unsigned long)inst->description,(unsigned long)"creates a file device for sim root folder");
					this->fileState 		= 210;
				}
				else {
					brdkStrCpy((unsigned long)inst->description,(unsigned long)"error calling DevUnlink. Flip enable to reset fb.");
					inst->status 				= this->DevUnlink_0.status;
					this->DevUnlink_0.enable 	= false;
					DevUnlink(&this->DevUnlink_0);
					this->fileState 			= 900;
				}
			}
			break;

		case 210:
			DevLink(&this->DevLink_0);
			if(this->DevLink_0.status != ERR_FUB_BUSY) {
				if(this->DevLink_0.status == ERR_OK) {
					this->DevUnlink_0.handle 	= this->DevLink_0.handle;
					this->DevLink_0.enable 		= false;
					DevLink(&this->DevLink_0);
					this->brdkFileCreateSubFolders_0.enable = true;
					brdkStrCpy((unsigned long)this->brdkFileCreateSubFolders_0.path,(unsigned long)sim->pcRootFolder);
					brdkStrCpy((unsigned long)this->brdkFileCreateSubFolders_0.fileDevice,this->DevLink_0.pDevice);
					brdkFileCreateSubFolders(&this->brdkFileCreateSubFolders_0);
					brdkStrCpy((unsigned long)inst->description,(unsigned long)"creates the needed folders");
					this->fileState 			= 220;
				}
				else {
					brdkStrCpy((unsigned long)inst->description,(unsigned long)"error calling DevLink. Flip enable to reset fb.");
					inst->status 				= this->DevLink_0.status;
					this->DevLink_0.enable 		= false;
					DevLink(&this->DevLink_0);
					this->fileState 			= 900;
				}
			}
			break;

		case 220:
			brdkFileCreateSubFolders(&this->brdkFileCreateSubFolders_0);
			if(this->brdkFileCreateSubFolders_0.done) {
				this->brdkFileCreateSubFolders_0.enable = false;
				brdkFileCreateSubFolders(&this->brdkFileCreateSubFolders_0);
				this->DevUnlink_0.enable 	= true;
				this->fileState				= 230;
			}
			else if(this->brdkFileCreateSubFolders_0.status != ERR_FUB_BUSY) {
				brdkStrCpy((unsigned long)inst->description,(unsigned long)"error calling brdkFileCreateSubFolders. Flip enable to reset fb.");
				inst->status 				= this->brdkFileCreateSubFolders_0.status;
				this->brdkFileCreateSubFolders_0.enable = false;
				brdkFileCreateSubFolders(&this->brdkFileCreateSubFolders_0);
				this->fileState 			= 900;
			}
			break;

		case 230:
			DevUnlink(&this->DevUnlink_0);
			if(this->DevUnlink_0.status != ERR_FUB_BUSY) {
				if(this->DevUnlink_0.status == ERR_OK) {
					this->DevUnlink_0.enable = false;
					DevUnlink(&this->DevUnlink_0);
					this->fileState 			= 0;
				}
				else {
					inst->status 				= this->DevUnlink_0.status;
					this->DevUnlink_0.enable 	= false;
					DevUnlink(&this->DevUnlink_0);
					brdkStrCpy((unsigned long)inst->description,(unsigned long)"error calling DevUnlink. Flip enable to reset fb.");
					this->fileState 			= 900;
				}
			}
			break;

		case 300: /* Remove device */
			DevUnlink(&this->DevUnlink_0);
			if(this->DevUnlink_0.status != ERR_FUB_BUSY) {
				if(this->DevUnlink_0.status == ERR_OK) {
					this->DevUnlink_0.enable = false;
					DevUnlink(&this->DevUnlink_0);
					this->activeHandles[this->fileIdx+1] = 0;

					this->DevLink_0.enable 	= true;
					if(setup->fileDevices[this->fileIdx].useUSB) this->DevLink_0.pDevice = (unsigned long)"ROOT";
					else 										 this->DevLink_0.pDevice = (unsigned long)"INTERNAL_ROOT";

					if(setup->fileDevices[this->fileIdx].useUSB) this->DevLink_0.pParam 	= buildParameterString((char*)&this->drive,(char*)&setup->fileDevices[this->fileIdx].path,(char*)&this->deviceParam);
					else{
						if(!DiagCpuIsSimulated()) getDrive(setup->plcDrive,this->driveInternal);
						else {
							getDrive(sim->pcHDDrive,this->driveInternal);
							brdkStrCat((unsigned long)this->driveInternal,(unsigned long)sim->pcRootFolder);
						}
						this->DevLink_0.pParam 	= buildParameterString((char*)&this->driveInternal,(char*)&setup->fileDevices[this->fileIdx].path,(char*)&this->deviceParam);
					}
					DevLink(&this->DevLink_0);
					brdkStrCpy((unsigned long)inst->description,(unsigned long)"switching to root device.");
					this->fileState = 310;
				}
				else {
					brdkStrCpy((unsigned long)inst->description,(unsigned long)"error calling DevUnlink. Flip enable to reset fb.");
					inst->status 				= this->DevUnlink_0.status;
					this->DevUnlink_0.enable 	= false;
					DevUnlink(&this->DevUnlink_0);
					this->fileState 			= 900;
				}
			}
			break;

		case 310: /* Switch to root device */
			DevLink(&this->DevLink_0);
			if(this->DevLink_0.status != ERR_FUB_BUSY) {
				if(this->DevLink_0.status == ERR_OK || this->DevLink_0.status == fiERR_DEVICE_ALREADY_EXIST) {
					this->DevLink_0.enable 	= false;
					DevLink(&this->DevLink_0);
					this->brdkFileCreateSubFolders_0.enable = true;
					brdkStrCpy((unsigned long)this->brdkFileCreateSubFolders_0.path,(unsigned long)setup->fileDevices[this->fileIdx].path);
					brdkStrCpy((unsigned long)this->brdkFileCreateSubFolders_0.fileDevice,(unsigned long)this->DevLink_0.pDevice);
					brdkFileCreateSubFolders(&this->brdkFileCreateSubFolders_0);
					brdkStrCpy((unsigned long)inst->description,(unsigned long)"creating the needed folder.");
					this->fileState 		= 320;
				}
				else{
					brdkStrCpy((unsigned long)inst->description,(unsigned long)"error changing the device. Flip enable to reset fb.");
					inst->status 			= this->DevLink_0.status;
					this->DevLink_0.enable 	= false;
					DevLink(&this->DevLink_0);
					this->fileState 		= 900;
				}
			}
			break;

		case 320: /* Create folder on device */
			brdkFileCreateSubFolders(&this->brdkFileCreateSubFolders_0);
			if(this->brdkFileCreateSubFolders_0.done) {
				this->brdkFileCreateSubFolders_0.enable = false;
				brdkFileCreateSubFolders(&this->brdkFileCreateSubFolders_0);
				this->DevLink_0.enable 	= true;
				this->DevLink_0.pDevice = (unsigned long)setup->fileDevices[this->fileIdx].name;
				if(setup->fileDevices[this->fileIdx].useUSB) this->DevLink_0.pParam 	= buildParameterString((char*)&this->drive,(char*)&setup->fileDevices[this->fileIdx].path,(char*)&this->deviceParam);
				else{
					if(!DiagCpuIsSimulated()) getDrive(setup->plcDrive,this->driveInternal);
					else {
						getDrive(sim->pcHDDrive,this->driveInternal);
						brdkStrCat((unsigned long)this->driveInternal,(unsigned long)sim->pcRootFolder);
					}
					this->DevLink_0.pParam 	= buildParameterString((char*)&this->driveInternal,(char*)&setup->fileDevices[this->fileIdx].path,(char*)&this->deviceParam);
				}
				DevLink(&this->DevLink_0);
				brdkStrCpy((unsigned long)inst->description,(unsigned long)"adding new device.");
				this->fileState 		= 330;

			}
			else if(this->brdkFileCreateSubFolders_0.status == fiERR_FILE_DEVICE) {
				if(DiagCpuIsSimulated()) {
//					this->DevUnlink_0.enable 	= true;
//					this->DevUnlink_0.handle 	= this->activeHandles[0];
//					this->activeHandles[0] 		= 0;
//					DevUnlink(&this->DevUnlink_0);
//					brdkStrCpy((unsigned long)this->brdkFileCreateSubFolders_0.path,(unsigned long)sim->pcRootFolder);
//
//					this->brdkFileCreateSubFolders_0.enable = false;
//					brdkFileCreateSubFolders(&this->brdkFileCreateSubFolders_0);
//
//					this->fileState 			= 400;
				}
				else {
					brdkStrCpy((unsigned long)inst->description,(unsigned long)"error calling brdkFileCreateSubFolders. Flip enable to reset fb.");
					inst->status 				= this->brdkFileCreateSubFolders_0.status;
					this->brdkFileCreateSubFolders_0.enable = false;
					brdkFileCreateSubFolders(&this->brdkFileCreateSubFolders_0);
					this->fileState 			= 900;
				}
			}
			else if(this->brdkFileCreateSubFolders_0.status != ERR_FUB_BUSY)
				brdkStrCpy((unsigned long)inst->description,(unsigned long)"error calling brdkFileCreateSubFolders. Check fb for error codes.");

			break;

		case 330: /* Switch to new device */
			DevLink(&this->DevLink_0);
			if(this->DevLink_0.status != ERR_FUB_BUSY) {
				if(this->DevLink_0.status == ERR_OK || this->DevLink_0.status == fiERR_DEVICE_ALREADY_EXIST) {
					this->activeHandles[this->fileIdx+1] = this->DevLink_0.handle;
					this->DevLink_0.enable 	= false;
					DevLink(&this->DevLink_0);
					inst->ready 				= true;
					brdkStrCpy((unsigned long)inst->description,(unsigned long)"all file devices are ready to use");
					this->fileState 			= 80;
				}
				else{
					brdkStrCpy((unsigned long)inst->description,(unsigned long)"error changing the device. Flip enable to reset fb.");
					inst->status 			= this->DevLink_0.status;
					this->DevLink_0.enable 	= false;
					DevLink(&this->DevLink_0);
					this->fileState 		= 900;
				}
			}
			break;

		case 900: /* error state */
			if(!inst->enable) {
				inst->status 	= 0;
				this->fileState = 0;
			}
			break;

	}

}
```

#### brdkFileWrite.c - Write data to a file.
```c
#include <brdkFile_func.h>

void brdkFileWrite(struct brdkFileWrite* inst) {
	brdk_file_write_internal_typ* this = (brdk_file_write_internal_typ*)&inst->internal;

	if(inst->enable) {

		switch(this->state) {

			case 0:
				inst->status = ERR_FUB_BUSY;
				this->FileCreate_0.enable 	= false;
				FileCreate(&this->FileCreate_0);
				this->FileCreate_0.enable 	= true;
				this->FileCreate_0.pDevice 	= inst->pFileDevice;
				this->FileCreate_0.pFile 	= inst->pFileName;
				this->state 				= 10;
				break;

			case 10:
				FileCreate(&this->FileCreate_0);
				switch(this->FileCreate_0.status) {

					case 0:	/* ERR_OK */
						this->FileWrite_0.enable 	= false;
						FileWrite(&this->FileWrite_0);
						this->FileWrite_0.enable 	= true;
						this->FileWrite_0.ident 	= this->FileCreate_0.ident;
						this->FileWrite_0.offset 	= 0;
						this->FileWrite_0.pSrc 		= inst->pData;
						this->FileWrite_0.len 		= inst->dataLength != 0 ? inst->dataLength : brdkStrLen(inst->pData);
						this->state 				= 40;
						break;

					case 20705: /* fiERR_EXIST  */
						if(!inst->overwrite) {
							this->FileOpen_0.enable 	= false;
							FileOpen(&this->FileOpen_0);
							this->FileOpen_0.enable 	= true;
							this->FileOpen_0.pDevice 	= inst->pFileDevice;
							this->FileOpen_0.pFile 		= inst->pFileName;
							this->FileOpen_0.mode 		= fiWRITE_ONLY;
							this->state 				= 20;
						}
						else {
							this->FileDelete_0.enable 	= false;
							FileDelete(&this->FileDelete_0);
							this->FileDelete_0.enable 	= true;
							this->FileDelete_0.pDevice 	= inst->pFileDevice;
							this->FileDelete_0.pName 	= inst->pFileName;
							this->state 				= 30;
						}
						break;

					case 65535: break;	/* ERR_FUB_BUSY */

					default:
						inst->status 				= this->FileCreate_0.status;
						this->state 				= 999;
						break;

				}
				break;

			case 20:
				FileOpen(&this->FileOpen_0);
				switch(this->FileOpen_0.status) {

					case 0:	/* ERR_OK */
						this->FileWrite_0.enable 	= false;
						FileWrite(&this->FileWrite_0);
						this->FileWrite_0.enable 	= true;
						this->FileWrite_0.ident 	= this->FileOpen_0.ident;
						this->FileWrite_0.offset 	= this->FileOpen_0.filelen;
						this->FileWrite_0.pSrc 		= inst->pData;			/* append the data tothe existing file */
						this->FileWrite_0.len 		= inst->dataLength != 0 ? inst->dataLength : brdkStrLen(inst->pData);
						this->state 				= 40;
						break;

					case 65535: break;	/* ERR_FUB_BUSY */

					default:
						inst->status 				= this->FileOpen_0.status;
						this->state 				= 999;
						break;

				}
				break;

			case 30:
				FileDelete(&this->FileDelete_0);
				switch(this->FileDelete_0.status) {

					case 0:	case 20708: /* ERR_OK - fiERR_FILE_NOT_FOUND */
						this->FileCreate_0.enable 	= false;
						FileCreate(&this->FileCreate_0);
						this->FileCreate_0.enable 	= true;
						this->FileCreate_0.pDevice 	= inst->pFileDevice;
						this->FileCreate_0.pFile 	= inst->pFileName;
						this->state 				= 10;
						break;

					case 65535: break;	/* ERR_FUB_BUSY */

					default:
						inst->status 				= this->FileDelete_0.status;
						this->state 				= 999;
						break;

				}
				break;

			case 40:
				FileWrite(&this->FileWrite_0);
				switch(this->FileWrite_0.status) {

					case 0:	/* ERR_OK */
						this->FileClose_0.enable 	= false;
						FileClose(&this->FileClose_0);
						this->FileClose_0.enable 	= true;
						this->FileClose_0.ident 	= this->FileWrite_0.ident;
						this->state 				= 50;
						break;

					case 65535: break;	/* ERR_FUB_BUSY */

					default:
						inst->status 				= this->FileWrite_0.status;
						this->state 				= 999;
						break;

				}
				break;

			case 50:
				FileClose(&this->FileClose_0);
				switch(this->FileClose_0.status) {

					case 0:	case 20721: /* ERR_OK - fiERR_FILE_NOT_OPENED */
						inst->status				= ERR_OK;
						this->state 				= 60;
						break;

					case 65535: break;	/* ERR_FUB_BUSY */

					default:
						inst->status 				= this->FileClose_0.status;
						this->state 				= 60;
						break;

				}
				break;

		}
	}
	else {
		inst->status				= ERR_FUB_ENABLE_FALSE;
		this->state 				= 0;
	}
}
```

#### brdkFileRead.c - Read data from a file.
```c
#include <brdkFile_func.h>

void brdkFileRead(struct brdkFileRead* inst) {
	brdk_file_read_internal_typ* this = (brdk_file_read_internal_typ*)&inst->internal;

	if(inst->enable) {
		switch(this->state) {

			case 0:	/* setup file open */
				inst->status = ERR_FUB_BUSY;
				this->FileOpen_0.enable 	= false;
				FileOpen(&this->FileOpen_0);
				this->FileOpen_0.enable 	= true;
				this->FileOpen_0.pDevice 	= inst->pFileDevice;
				this->FileOpen_0.pFile 		= inst->pFileName;
				this->FileOpen_0.mode 		= fiREAD_ONLY;
				this->state 				= 10;
				break;

			case 10: /* call file open */
				FileOpen(&this->FileOpen_0);
				switch(this->FileOpen_0.status) {

					case 0:	/* ERR_OK */
						this->FileRead_0.enable 	= false;
						FileRead(&this->FileRead_0);
						this->FileRead_0.enable 	= true;
						this->FileRead_0.ident 		= this->FileOpen_0.ident;
						this->FileRead_0.offset 	= 0;
						this->FileRead_0.pDest 		= inst->pData;
						if(this->FileOpen_0.filelen < inst->dataLength) this->FileRead_0.len = this->FileOpen_0.filelen;
						else this->FileRead_0.len 	= inst->dataLength;
						this->state 				= 20;
						break;

					case 65535: break;	/* ERR_FUB_BUSY */

					default:
						inst->status 				= this->FileOpen_0.status;
						this->state 				= 999;
						break;

				}
				break;

			case 20: /* call file read */
				FileRead(&this->FileRead_0);
				switch(this->FileRead_0.status) {

					case 0:	/* ERR_OK */
						this->FileClose_0.enable 	= false;
						FileClose(&this->FileClose_0);
						this->FileClose_0.enable 	= true;
						this->FileClose_0.ident 	= this->FileRead_0.ident;
						this->state 				= 30;
						break;

					case 65535: break;	/* ERR_FUB_BUSY */

					default:
						inst->status 				= this->FileRead_0.status;
						this->state 				= 999;
						break;

				}
				break;

			case 30: /* call file close */
				FileClose(&this->FileClose_0);
				switch(this->FileClose_0.status) {

					case 0:	case 20721: /* ERR_OK - fiERR_FILE_NOT_OPENED */
						inst->readLength			= this->FileOpen_0.filelen;
						inst->status				= ERR_OK;
						this->state 				= 40;
						break;

					case 65535: break;	/* ERR_FUB_BUSY */

					default:
						inst->status 				= this->FileClose_0.status;
						this->state 				= 999;
						break;

				}
				break;

		}

	}
	else {
		inst->status				= ERR_FUB_ENABLE_FALSE;
		inst->readLength			= 0;
		this->state 				= 0;
	}
}
```

#### brdkFile_func.c - Internal functions for library.
```c
#include <brdkFile_func.h>

unsigned long buildParameterString(char* pDrive,char* pPath, char* pDeviceParam) {
	brdkStrCpy((unsigned long)pDeviceParam,(unsigned long)"/DEVICE=\"");
	brdkStrCat((unsigned long)pDeviceParam,(unsigned long)pDrive);
	brdkStrCat((unsigned long)pDeviceParam,(unsigned long)"\\");
	if(pPath[0] != 0) {
		brdkStrReplace((unsigned long)pPath,(unsigned long)"/",(unsigned long)"\\");	/* replace any frontslash with backslash */
		brdkStrCat((unsigned long)pDeviceParam,(unsigned long)pPath);
	}
	brdkStrCat((unsigned long)pDeviceParam,(unsigned long)"\"");
	return (unsigned long)pDeviceParam;
}

char* getDrive(brdk_file_drive_typ drive, char* pDrive) {
	switch(drive) {
		case C_DRIVE: brdkStrCpy((unsigned long)pDrive,(unsigned long)"C:\\"); break;
		case D_DRIVE: brdkStrCpy((unsigned long)pDrive,(unsigned long)"D:\\"); break;
		case E_DRIVE: brdkStrCpy((unsigned long)pDrive,(unsigned long)"E:\\"); break;
		case F_DRIVE: brdkStrCpy((unsigned long)pDrive,(unsigned long)"F:\\"); break;
		case G_DRIVE: brdkStrCpy((unsigned long)pDrive,(unsigned long)"G:\\"); break;
	}
	return pDrive;
}

signed long splitFolderPath(char* pDestination, char* pSource) {
	int idx = 0;
	signed long pos = -1;
	if(pSource[idx] != 0) {
		pos = brdkStrIndexOf((unsigned long)&pSource[idx],(unsigned long)"\\",BRDK_STR_LEFT_SEARCH);
		if(pos > -1) {
			brdkStrMemCpy((unsigned long)pDestination,(unsigned long)&pSource[idx],(unsigned long)++pos);
			pDestination[pos] = 0;
		}
	}
	return pos;
}
```

- CHANGELOG - brdkFile change log file (not shown)

### Program Logical/SM/StateMachine

#### Main.st
```iecst
PROGRAM _INIT

	gStateMachine.status.state 			:= STATE_INITIALIZE;
	gStateMachine.status.stateOld 		:= gStateMachine.status.state;

	gStateMachine.status.stateChangeTimeout := FALSE;

	gIsSimulation 						:= DiagCpuIsSimulated();
	//gIsSimulation 	:= TRUE;

	(* Initialize the strings for the instructions *)
	initInstructions;

	initForceIO;

	TON_stateChange.PT 			:= T#500ms;
	this.TON_initialization.PT 	:= T#3s;
	TON_stateTimeout.PT 		:= T#15s;

END_PROGRAM

PROGRAM _CYCLIC
	(* Instruction to tell the driver what to do *)
	instruction;

	forceIO;

	// Handle state timeout
	TON_stateTimeout.IN := gStateMachine.status.state = STATE_ENABLING_SC OR gStateMachine.status.state = STATE_PRECHARGING;
	TON_stateTimeout();
	gStateMachine.status.stateChangeTimeout := TON_stateTimeout.Q;

	// Handle delay between state changes
	changeStateDelay;

	IF gEventLog.resetEventLog THEN
		resetEventLog;
	END_IF;

	CASE gStateMachine.status.state OF
		(* The car startsup in this state. It controls the startup routine *)
		STATE_INITIALIZE:
			gStateMachine.status.stateName := 'Initialize';
			stateInit;
			stateChangeInit;

		(* 	Idle state where the car is when it is OK for driving but is waiting for start commands.
			The car enters this state when the startup routine is done and after a broken safety chain is closed *)
		STATE_IDLE:
			gStateMachine.status.stateName := 'Idle';
			stateIdle;
			stateChangeIdle;

		(* The AMS is opening the SC *)
		STATE_ENABLING_SC:
			gStateMachine.status.stateName := 'Enabling Shutdown Circuit';
			stateEnablingSC;
			stateChangeEnablingSC;

		(* The last part of the safety chain is enabled and the safety chain is fully closed *)
		STATE_SC_ENABLED:
			gStateMachine.status.stateName := 'Shutdown Circuit Enabled';
			stateSCEnabled;
			stateChangeSCEnabled;

		(* The SC is currently charging *)
		STATE_PRECHARGING:
			gStateMachine.status.stateName := 'Precharging';
			statePrecharging;
			stateChangePrecharging;

		(* The AIRs are closed and precharging is enabled *)
		STATE_TRACTIVE:
			gStateMachine.status.stateName := 'Tractive';
			stateTractive;
			stateChangeTractive;

		(* The car is in a driving state and pressing the torque pedal propels the car *)
		STATE_DRIVE:
			gStateMachine.status.stateName := 'Drive';
			stateDrive;
			stateChangeDrive;

		(* One or more elements of the safety chain are broken *)
		STATE_ERROR:
			gStateMachine.status.stateName := 'Error';
			stateError;
			stateChangeError;
		ELSE
	END_CASE

	// Log state change event
	IF gStateMachine.status.stateName <> gStateMachine.status.stateNameOld THEN
		gEventLog.newEventString := 'State changed to: ';
		strcat(ADR(gEventLog.newEventString),ADR(gStateMachine.status.stateName));
		logEvent;
	END_IF;
	gStateMachine.status.stateNameOld := gStateMachine.status.stateName;

END_PROGRAM

PROGRAM _EXIT

END_PROGRAM
```

#### Program Logical/SM/StateMachine/functions

##### instruction.st
```iecst
ACTION initInstructions:
	this.instructionList[INST_INITIALIZING] 			:= 'Initializing';
	this.instructionList[INST_PRESS_SAFETY_BUTTON] 		:= 'Press Safety Button';
	this.instructionList[INST_SC_NOT_ENABLED]			:= 'Wait for SC to be Enabled';
	this.instructionList[INST_PRESS_TRACTIVE_BUTTON] 	:= 'Press Tractive Button';
	this.instructionList[INST_AMS_NOT_READY]			:= 'Wait for AMS to be Ready';
	this.instructionList[INST_PRESS_BRAKE] 				:= 'Press Brake Predal';
	this.instructionList[INST_TORQUE_PEDAL_FAULT] 		:= 'Torque Pedal Fault';
	this.instructionList[INST_PRE_CHARGING] 			:= 'Pre-Charging. Wait';
	this.instructionList[INST_PRESS_DRIVE_BUTTON] 		:= 'Press Drive Button';
	this.instructionList[INST_FIX_ERROR] 				:= 'Remove Error';
	this.instructionList[INST_CLOSE_SAFETY_CHAIN] 		:= 'Close Shutdown Circuit';
	this.instructionList[INST_IN_DRIVE] 				:= 'To Exit Drive: Press Shutdown Button';
END_ACTION

ACTION instruction:
	IF gStateMachine.status.instructionIndex = INST_CLOSE_SAFETY_CHAIN THEN
		gStateMachine.status.instruction := CONCAT(this.instructionList[INST_CLOSE_SAFETY_CHAIN], ' at: ');
		gStateMachine.status.instruction := CONCAT(gStateMachine.status.instruction, gSafetyChain.status.scErrorString);

		ELSE
			gStateMachine.status.instruction := this.instructionList[gStateMachine.status.instructionIndex];

		END_IF
END_ACTION
```

#### Program Logical/SM/StateMachine/states

##### statePrecharging.st
```iecst
(* State Ready *)
ACTION statePrecharging:

END_ACTION

(* State Ready *)
ACTION stateChangePrecharging:
	IF gStateMachine.status.stateChangeAllowed THEN
		(* Update Instruction Index *)
		gStateMachine.status.instructionIndex := INST_PRE_CHARGING;

		IF gAMS.status.prechargingDone THEN
			gStateMachine.status.state := STATE_TRACTIVE;
		END_IF

		IF gStateMachine.status.stateChangeTimeout THEN
			gAMS.cmd.abort 				:= TRUE;
			gStateMachine.status.state 	:= STATE_IDLE;
		END_IF;

		(* If safety chain is broken go to state 'stateError' *)
		IF NOT gSafetyChain.status.scOKPersistent THEN
			gStateMachine.status.state 	:= STATE_ERROR;
			gAMS.cmd.abort 				:= TRUE;
		END_IF
	END_IF;
END_ACTION
```

##### stateTractive.st
```iecst
(* State Tractive *)
ACTION stateTractive:
	// Wait for a command to either go to drive or charging

END_ACTION

	(* Conditions for state change for STATE_OPENING_RELAYS *)
ACTION stateChangeTractive:
	IF gStateMachine.status.stateChangeAllowed THEN

		(* If precharge is done and brake pressure is over threshold and drive button pressed change state to 'stateDrive'  *)

		(* If brakes are pressed *)
		IF 	gBraking.status.softBraking THEN
			(* No torque pedal critical error *)
			IF  NOT gTorqueSensor.status.criticalError AND gTorqueSensor.status.torquePercentage < 10 THEN
				(* Wait for AMS to be ready *)
				//IF gAMS.status.amsState = AMS_STATE_TC_ENABLED OR gAMS.status.amsState = AMS_STATE_DRIVE THEN
				IF gORION.state = PRECHARGING_DONE THEN
					(* Update instruction string. Press drive button *)
					gStateMachine.status.instructionIndex := INST_PRESS_DRIVE_BUTTON;

					(* Mark that the car is ready to go into drive *)
					gStateMachine.status.readyForStateDrive := TRUE;

					(* Pushing the drive button will set the car in state drive *)
					IF EDGEPOS(gDashboard.inputs.di_buttonDrive) THEN

						gStateMachine.status.state 	:= STATE_DRIVE;
						gAMS.cmd.enterDrive 		:= TRUE;

						(* If the PLC is simulated reset the button *)
						IF gIsSimulation THEN
							gDashboard.inputs.di_buttonDrive := FALSE;
						END_IF
					END_IF
				ELSE
					(* Wait for AMS to be ready *)
					gStateMachine.status.instructionIndex := INST_AMS_NOT_READY;
				END_IF;
			ELSE
				(* Update instruction string. Torque sensors out of range *)
				gStateMachine.status.instructionIndex := INST_TORQUE_PEDAL_FAULT;
			END_IF
		ELSE
			(* Update instruction string. Press brake *)
			gStateMachine.status.instructionIndex := INST_PRESS_BRAKE;
		END_IF

		(* If safety chain is broken go to state 'stateError' *)
		IF NOT gSafetyChain.status.scOKPersistent THEN
			gStateMachine.status.state 	:= STATE_ERROR;
			gAMS.cmd.abort 				:= TRUE;
		END_IF

	END_IF;

END_ACTION
```

### globalSafetyChain.typ
```iecst
TYPE
	gSafetyChain_cmd_typ : 	STRUCT
		di_LVMS_OK : BOOL;
		di_supply : BOOL;
		di_shutdownCockpit_OK : BOOL;
		di_BOTS_OK : BOOL;
		di_inertiaSwitch_OK : BOOL;
		di_shutdownLeft_OK : BOOL;
		di_shutdownRight_OK : BOOL;
		di_interlockWheelFR_OK : BOOL;
		di_interlockWheelFL_OK : BOOL;
		di_interlockWheelRR_OK : BOOL;
		di_interlockWheelRL_OK : BOOL;
		di_interlockHVDC_OK : BOOL;
		di_IMD_OK : BOOL;
		di_AMS_OK : BOOL;
		di_TS_Container : BOOL;
		di_BSPD_OK : BOOL;
		di_interlockHVD_OK : BOOL;
		di_interlockMotorRR_OK : BOOL;
		di_interlockMotorRL_OK : BOOL;
		di_interlockMotorFR_OK : BOOL;
		di_interlockMotorFL_OK : BOOL;
		di_interlockTSMP_OK : BOOL;
		di_TSMS_OK : BOOL;
	END_STRUCT;
	gSafetyChain_typ : 	STRUCT
		status : gSafetyChain_status_typ;
		outputs : gSafetyChain_outputs_typ;
		data : gSafetyChain_data_typ;
		inputs : gSafetyChain_inputs_typ;
		cmd : gSafetyChain_cmd_typ;
	END_STRUCT;
	gSafetyChain_status_typ : 	STRUCT
		scOK_notEnabled : BOOL;
		scOK_usint : USINT;
		scOKPersistent : BOOL;
		scOK : BOOL;
		scErrorIndex : USINT;
		sc : ARRAY[0..MAX_SC_ELEMENTS]OF BOOL;
		scErrorStrings : ARRAY[0..MAX_SC_ELEMENTS]OF STRING[80];
		scErrorString : STRING[80];
		safetyChainEnabled : BOOL;
	END_STRUCT;
	gSafetyChain_inputs_typ : 	STRUCT
		di_LVMS_OK : BOOL;
		di_supply : BOOL;
		di_shutdownCockpit_OK : BOOL;
		di_BOTS_OK : BOOL;
		di_inertiaSwitch_OK : BOOL;
		di_shutdownLeft_OK : BOOL;
		di_shutdownRight_OK : BOOL;
		di_interlockWheelFR_OK : BOOL;
		di_interlockWheelFL_OK : BOOL;
		di_interlockWheelRR_OK : BOOL;
		di_interlockWheelRL_OK : BOOL;
		interlockHVDC_OK : BOOL;
		IMD_OK : BOOL;
		AMS_OK : BOOL;
		di_TS_Container : BOOL;
		di_BSPD_OK : BOOL;
		di_interlockHVD_OK : BOOL;
		di_interlockMotorRR_OK : BOOL;
		di_interlockMotorRL_OK : BOOL;
		di_interlockMotorFR_OK : BOOL;
		di_interlockMotorFL_OK : BOOL;
		di_interlockTSMP_OK : BOOL;
		di_interlockMotorConBoxFR_OK : BOOL;
		di_interlockMotorConBoxFL_OK : BOOL;
		di_TSMS_OK : BOOL;
	END_STRUCT;
	gSafetyChain_outputs_typ : 	STRUCT
		dummy : BOOL;
	END_STRUCT;
	gSafetyChain_data_typ : 	STRUCT
		dummy : USINT;
	END_STRUCT;
END_TYPE
```

### Program Logical/SC/SafetyChain

#### scStrings.st
```iecst
(* Write SC error names into array *)
ACTION scStrings:
	gSafetyChain.status.scErrorStrings[0] := 'Low Voltage Master Switch';
	gSafetyChain.status.scErrorStrings[1] := 'Supply';
	gSafetyChain.status.scErrorStrings[2] := 'Cockpit Shutdown Button';
	gSafetyChain.status.scErrorStrings[3] := 'BOTS';
	gSafetyChain.status.scErrorStrings[4] := 'Inertia Switch';
	gSafetyChain.status.scErrorStrings[5] := 'Left Shutdown Button';
	gSafetyChain.status.scErrorStrings[6] := 'Right Shutodwn Button';
	gSafetyChain.status.scErrorStrings[7] := 'FR Wheel Interlock';
	gSafetyChain.status.scErrorStrings[8] := 'FL Wheel Interlock';
	gSafetyChain.status.scErrorStrings[9] := 'RR Wheel Interlock';
	gSafetyChain.status.scErrorStrings[10] := 'RL Wheel Interlock';
	gSafetyChain.status.scErrorStrings[11] := 'HVDC Interlock';
	gSafetyChain.status.scErrorStrings[12] := 'IMD';
	gSafetyChain.status.scErrorStrings[13] := 'AMS';
	gSafetyChain.status.scErrorStrings[14] := 'TS container';
	gSafetyChain.status.scErrorStrings[15] := 'BSPD';
	gSafetyChain.status.scErrorStrings[16] := 'HVD Interlock';
	gSafetyChain.status.scErrorStrings[17] := 'TS Container interlocks';
	gSafetyChain.status.scErrorStrings[18] := 'TS Container interlocks';
	gSafetyChain.status.scErrorStrings[19] := 'TS Container interlocks';
	gSafetyChain.status.scErrorStrings[20] := 'TS Container interlocks';
	gSafetyChain.status.scErrorStrings[21] := 'TSMP or MotorConBox';
	gSafetyChain.status.scErrorStrings[22] := 'TSMP or MotorConBox';
	gSafetyChain.status.scErrorStrings[23] := 'TSMP or MotorConBox';
//	gSafetyChain.status.scErrorStrings[15] := 'FR Motor Interlock';
//	gSafetyChain.status.scErrorStrings[16] := 'FL Motor Interlock';
//	gSafetyChain.status.scErrorStrings[17] := 'RR Motor Interlock';
//	gSafetyChain.status.scErrorStrings[18] := 'RL Motor Interlock';
//	gSafetyChain.status.scErrorStrings[19] := 'TSMPs Interlock';
	gSafetyChain.status.scErrorStrings[24] := 'Tractive System Master Switch';
	gSafetyChain.status.scErrorStrings[25] := 'Shutdown Circuit Enable';
	gSafetyChain.status.scErrorStrings[26] := ' ';
END_ACTION
```

#### scUpdate.st
```iecst
(* Write SC values into array *)
ACTION scUpdate:
	(* Collect inputs that are in groups *)
//	gSafetyChain.inputs.di_interlockMotorFR_OK := gSafetyChain.inputs.di_interlockTSMP_OK;	// 'FR Motor Interlock';
//	gSafetyChain.inputs.di_interlockMotorFL_OK := gSafetyChain.inputs.di_interlockTSMP_OK;	// 'FL Motor Interlock';
//	gSafetyChain.inputs.di_interlockMotorRR_OK := gSafetyChain.inputs.di_interlockTSMP_OK;	// 'RR Motor Interlock';
//	gSafetyChain.inputs.di_interlockMotorRL_OK := gSafetyChain.inputs.di_interlockTSMP_OK;	// 'RL Motor Interlock';

	// All 4 motor interlocks are dependant on the input from the RL motor
	gSafetyChain.inputs.di_interlockMotorFR_OK := gSafetyChain.inputs.di_interlockMotorRL_OK;	// 'FR Motor Interlock';
	gSafetyChain.inputs.di_interlockMotorFL_OK := gSafetyChain.inputs.di_interlockMotorRL_OK;	// 'FL Motor Interlock';
	gSafetyChain.inputs.di_interlockMotorRR_OK := gSafetyChain.inputs.di_interlockMotorRL_OK;	// 'RR Motor Interlock';

	// Connection boxes for front motors interlocks dependent on signal from TSMP
	gSafetyChain.inputs.di_interlockMotorConBoxFL_OK := gSafetyChain.inputs.di_interlockTSMP_OK;	// 'FL Motor Connection Box Interlock';
	gSafetyChain.inputs.di_interlockMotorConBoxFR_OK := gSafetyChain.inputs.di_interlockTSMP_OK;	// 'FR Motor Connection Box Interlock';

	(* Write safety chain values to array *)
	gSafetyChain.status.sc[0]  := gSafetyChain.inputs.di_LVMS_OK; 				// 'Low Voltage Master Switch';
	gSafetyChain.status.sc[1]  := gSafetyChain.inputs.di_supply;				// 'Supply'
	gSafetyChain.status.sc[2]  := gSafetyChain.inputs.di_shutdownCockpit_OK; 	// 'Cockpit Shutdown Button';
	gSafetyChain.status.sc[3]  := gSafetyChain.inputs.di_BOTS_OK;				// 'BOTS';
	gSafetyChain.status.sc[4]  := gSafetyChain.inputs.di_inertiaSwitch_OK;		// 'Intertia Switch';
	gSafetyChain.status.sc[5]  := gSafetyChain.inputs.di_shutdownLeft_OK; 		//'Left Shutdown Button';
	gSafetyChain.status.sc[6]  := gSafetyChain.inputs.di_shutdownRight_OK;		// 'Right Shutodwn Button';
	gSafetyChain.status.sc[7]  := gSafetyChain.inputs.di_interlockWheelFR_OK;	// 'FR Wheel Interlock';
	gSafetyChain.status.sc[8]  := gSafetyChain.inputs.di_interlockWheelFL_OK;	// 'FL Wheel Interlock';
	gSafetyChain.status.sc[9]  := gSafetyChain.inputs.di_interlockWheelRR_OK;	// 'RR Wheel Interlock';
	gSafetyChain.status.sc[10] := gSafetyChain.inputs.di_interlockWheelRL_OK;	// 'RL Wheel Interlock';
	gSafetyChain.status.sc[11] := gSafetyChain.inputs.interlockHVDC_OK;			// 'HV DC Interlock';
	gSafetyChain.status.sc[12] := gSafetyChain.inputs.IMD_OK;					// 'IMD';
	gSafetyChain.status.sc[13] := gSafetyChain.inputs.AMS_OK;					// 'AMS';
	gSafetyChain.status.sc[14] := gSafetyChain.inputs.di_TS_Container;			// 'TS Container';
	gSafetyChain.status.sc[15] := gSafetyChain.inputs.di_BSPD_OK;				// 'BSPD';
	gSafetyChain.status.sc[16] := gSafetyChain.inputs.di_interlockHVD_OK;		// 'HVD Interlock';
	gSafetyChain.status.sc[17] := gSafetyChain.inputs.di_interlockMotorFR_OK;	// 'FR Motor Interlock';
	gSafetyChain.status.sc[18] := gSafetyChain.inputs.di_interlockMotorFL_OK;	// 'FL Motor Interlock';
	gSafetyChain.status.sc[19] := gSafetyChain.inputs.di_interlockMotorRR_OK;	// 'RR Motor Interlock';
	gSafetyChain.status.sc[20] := gSafetyChain.inputs.di_interlockMotorRL_OK;	// 'RL Motor Interlock';
	gSafetyChain.status.sc[21] := gSafetyChain.inputs.di_interlockMotorConBoxFL_OK;	// 'FL Motor ConBox Interlock';
	gSafetyChain.status.sc[22] := gSafetyChain.inputs.di_interlockMotorConBoxFR_OK;	// 'FR Motor ConBox Interlock';
	gSafetyChain.status.sc[23] := gSafetyChain.inputs.di_interlockTSMP_OK;		// 'TSMP Interlock';
	gSafetyChain.status.sc[24] := gSafetyChain.inputs.di_TSMS_OK;				// 'Tractive System Master Switch';
	gSafetyChain.status.sc[25] := gAMS.status.scEnabled;						// 'Safety Chain Enable';
	gSafetyChain.status.sc[26] := FALSE;
END_ACTION
```

### globalAMS.typ
```iecst
TYPE
	gAMS_cmd_typ : 	STRUCT
		chargingPrescalerAmp : REAL;
		chargingPrescalerPercent : USINT;
		bankCount : USINT;
		mpo1 : USINT;
		mpo2 : USINT;
		mpo3 : USINT;
		mpe : USINT;
		commandId : USINT;
		startPrecharge : BOOL;
		enableSC : BOOL;
		enterDrive : BOOL;
		abort : BOOL;
	END_STRUCT;
	gAMS_data_history_typ : 	STRUCT
		actPower : ARRAY[0..999]OF REAL;
		actCurrent : ARRAY[0..999]OF REAL;
		actSoc : ARRAY[0..999]OF REAL;
		actVoltage : ARRAY[0..999]OF REAL;
	END_STRUCT;
	gAMS_data_typ : 	STRUCT
		stateOfCharge : REAL;
		outputCurrent : REAL;
		chargeCurrent : REAL;
		batteryVoltage : REAL;
		cellTempMax : REAL;
		cellVoltageMax : ARRAY[0..4]OF REAL;
		cellVoltageMin : ARRAY[0..4]OF REAL;
		bankTemperatureMax : ARRAY[0..4]OF REAL;
		bankTemperatureMin : ARRAY[0..4]OF REAL;
		bankResistorTemperatureMax : ARRAY[0..4]OF REAL;
		bankResistorTemperatureMin : ARRAY[0..4]OF REAL;
		history : gAMS_data_history_typ;
		packPower : REAL;
		cellVoltageMinOrion : REAL;
		batteryTempMax : REAL;
	END_STRUCT;
	gAMS_inputs_typ : 	STRUCT
		dummy : USINT;
	END_STRUCT;
	gAMS_outputs_typ : 	STRUCT
		com_idle : BOOL;
		com_sc_enable : BOOL;
		com_precharge : BOOL;
		com_drive : BOOL;
		com_charge : BOOL;
		com_resetShunt : BOOL;
	END_STRUCT;
	gAMS_status_bank_typ : 	STRUCT
		bankVoltage : REAL;
		resistorTemperature : ARRAY[0..13]OF REAL;
		temperatures : ARRAY[0..9]OF REAL;
		cellVoltage : ARRAY[0..27]OF REAL;
	END_STRUCT;
	gAMS_status_error_typ : 	STRUCT
		errorTimers : ARRAY[0..21]OF TON;
		amsError : BOOL;
		imdError : BOOL;
		hvdcInterlockError : BOOL;
		tempWarn : BOOL;
		voltWarn : BOOL;
		precharge : BOOL;
		airMinus : BOOL;
		airPlus : BOOL;
		lowVoltage : BOOL;
		highVoltage : BOOL;
		lowTemp : BOOL;
		highTemp : BOOL;
		ltc6813Com : BOOL;
		shuntCom : BOOL;
		openSc : BOOL;
		closeSc : BOOL;
		openAirMinus : BOOL;
		closeAirMinus : BOOL;
		openAirPlus : BOOL;
		closeAirPlus : BOOL;
		openPrePlus : BOOL;
		closePrePlus : BOOL;
		preTimeout : BOOL;
		unexpectedChargeRate : BOOL;
		bankCountMismatch : BOOL;
		unexpectedTsCurrent : BOOL;
		relayFailed : BOOL;
		scBroken : BOOL;
		unfitChargeVoltage : BOOL;
		monitorError : BOOL;
	END_STRUCT;
	gAMS_status_pack_typ : 	STRUCT
		packVoltage : REAL;
		resistorTemperature : ARRAY[0..69]OF REAL;
		temperatures : ARRAY[0..49]OF REAL;
		InstantCellVoltage : ARRAY[0..179]OF REAL;
		cellTempMax : SINT;
		cellVoltage : ARRAY[0..179]OF REAL;
	END_STRUCT;
	gAMS_status_failsafe_typ : 	STRUCT
		failsafeStatus : UINT;
	END_STRUCT;
	gAMS_status_relay_typ : 	STRUCT
		dischargeRelayEnabled : BOOL;
		chargeRelayEnabled : BOOL;
		chargerSafetyEnabled : BOOL;
		malfunctionIndicatorActive : BOOL;
		MPI1SignalStatus : BOOL;
		alwaysOnSignalStatus : BOOL;
		isReadyInputStatus : BOOL;
		isChargingInputStatus : BOOL;
		MPI2SignalStatus : BOOL;
		MPI3SignalStatus : BOOL;
		chargeModeStatus : BOOL;
		MPO2SignalStatus : BOOL;
		MPO3SignalStatus : BOOL;
		MPO4SignalStatus : BOOL;
		MPEnableSignalStatus : BOOL;
		MPO1SignalStatus : BOOL;
		relayState : UINT;
	END_STRUCT;
	gAMS_status_typ : 	STRUCT
		ok : BOOL;
		pack : gAMS_status_pack_typ;
		bank : ARRAY[0..4]OF gAMS_status_bank_typ;
		error : gAMS_status_error_typ;
		hasError : BOOL;
		amsBankCount : USINT;
		amsStateName : STRING[80];
		amsState : USINT;
		amsTurnedOnCharger : BOOL;
		scEnabled : BOOL;
		highPowerWarning : BOOL;
		highPowerError : BOOL;
		disconnected : BOOL;
		prechargingDone : BOOL;
		Counter : USINT;
		relayState : gAMS_status_relay_typ;
		failsafeStatus : gAMS_status_failsafe_typ;
		DTC1Status : UINT;
		DTC2Status : UINT;
		RelayError : USINT;
		errorInfo : STRING[80];
	END_STRUCT;
	gAMS_typ : 	STRUCT
		status : gAMS_status_typ;
		outputs : gAMS_outputs_typ;
		data : gAMS_data_typ;
		inputs : gAMS_inputs_typ;
		cmd : gAMS_cmd_typ;
	END_STRUCT;
END_TYPE
```

### globalORION.var
```iecst
VAR
	TON_prechargeDisableDrive : TON;
	gORION : gORION_typ;
END_VAR
```

### globalShunt.var
```iecst
VAR
	gShunt : gShunt_typ;
END_VAR
```

### Program Logical/AMS_and_Shunt/AMS (IEC)

#### Main.st
```iecst
PROGRAM _INIT

	gAMS.data.outputCurrent := 0;
	gAMS.data.stateOfCharge := 0;
//	gAMS.data.totalPower 	:= 0;
//	gAMS.data.totalPowerMax := 0;  // Reset variable used to keep track of the maximum power used

	powerHistoryInverval 		:= T#10ms;
	currentHistoryInverval 		:= T#20ms;
	socHistoryInverval			:= T#500ms;
	voltageHistoryInverval  	:= T#100ms;
	gORION.data.TON_counter.PT	:= T#1s;

	constant.fullBatteryCapacityAh  := 12.5;
	constant.fullBatteryCapacitykWh := 6.475;

	constant.chargingCurrentMax := 12.5;
	gAMS.cmd.chargingPrescalerAmp := constant.chargingCurrentMax;

	gAMS.cmd.bankCount := 5;

	errorsInit_action;

END_PROGRAM

PROGRAM _CYCLIC

	states;
	orionErrorAction;
	error_action;

	gAMS.data.chargeCurrent := - gAMS.data.outputCurrent;

//	gAMS.data.batteryVoltage := gAMS.status.bank[0].bankVoltage + gAMS.status.bank[1].bankVoltage +
//								gAMS.status.bank[2].bankVoltage + gAMS.status.bank[3].bankVoltage + gAMS.status.bank[4].bankVoltage;

	gAMS.data.batteryTempMax := MAX(gAMS.data.bankTemperatureMax[0], gAMS.data.bankTemperatureMax[1], gAMS.data.bankTemperatureMax[2],
							 gAMS.data.bankTemperatureMax[3]);

	gAMS.cmd.chargingPrescalerPercent := LIMIT(0, REAL_TO_USINT((gAMS.cmd.chargingPrescalerAmp / constant.chargingCurrentMax) * 100), 100);

	powerMonitoring;

	(* Determine if AMS has an error or not *)
	gAMS.status.ok 	 := (NOT gAMS.status.disconnected) AND (NOT (gAMS.status.amsStateName = 'ERROR')) AND (NOT gAMS.status.hasError);
	gShunt.status.ok := NOT gShunt.status.disconnected;

//	gAMS.data.stateOfCharge := ((constant.fullBatteryCapacitykWh-gShunt.data.actPowerKWH) / constant.fullBatteryCapacitykWh) * 100.00;

	// Calculating the voltage of each bank
	FOR j := 0 TO BANK_COUNT-1 DO
		k := CELL_COUNT*j;
		tmpVoltage := 0;
		FOR i := 0 TO CELL_COUNT-1 DO
			// gAMS.status.bank[j].cellVoltage[i] := gAMS.status.pack.cellVoltage[i + k];
			tmpVoltage := tmpVoltage + gAMS.status.bank[j].cellVoltage[i];
		END_FOR;
		gAMS.status.bank[j].bankVoltage := tmpVoltage;
	END_FOR

	FOR j := 0 TO BANK_COUNT-1 DO
		// Max voltage
		tmpVoltageMax := 0;
		FOR i := 0 TO CELL_COUNT-1 DO
			IF gAMS.status.bank[j].cellVoltage[i] > tmpVoltageMax THEN
				tmpVoltageMax := gAMS.status.bank[j].cellVoltage[i];
			END_IF;
		END_FOR;
		gAMS.data.cellVoltageMax[j] := tmpVoltageMax;

		// Min voltage
		tmpVoltageMin := 10000;
		FOR i := 0 TO CELL_COUNT-1 DO
			IF gAMS.status.bank[j].cellVoltage[i] < tmpVoltageMin THEN
				tmpVoltageMin := gAMS.status.bank[j].cellVoltage[i];
			END_IF;
		END_FOR;
		gAMS.data.cellVoltageMin[j] := tmpVoltageMin;

		// Max temperature
		tmpTemperatureMax := 0;
		FOR i := 0 TO TEMPERATURE_COUNT-1 DO
			IF gAMS.status.bank[j].temperatures[i] > tmpTemperatureMax THEN
				tmpTemperatureMax := gAMS.status.bank[j].temperatures[i];
			END_IF;
		END_FOR;
		gAMS.data.bankTemperatureMax[j] := tmpTemperatureMax;

		// Min temperature
		tmpTemperatureMin := 10000;
		FOR i := 0 TO TEMPERATURE_COUNT-1 DO
			IF gAMS.status.bank[j].temperatures[i] < tmpTemperatureMin THEN
				tmpTemperatureMin := gAMS.status.bank[j].temperatures[i];
			END_IF;
		END_FOR;
		gAMS.data.bankTemperatureMin[j] := tmpTemperatureMin;

		// Max resistor temperature
		tmpTemperatureMax := 0;
		FOR i := 0 TO RESISTOR_COUNT-1 DO
			IF gAMS.status.bank[j].resistorTemperature[i] > tmpTemperatureMax THEN
				tmpTemperatureMax := gAMS.status.bank[j].resistorTemperature[i];
			END_IF;
		END_FOR;
		gAMS.data.bankResistorTemperatureMax[j] := tmpTemperatureMax;

		// Min temperature
		tmpTemperatureMin := 10000;
		FOR i := 0 TO RESISTOR_COUNT-1 DO
			IF gAMS.status.bank[j].resistorTemperature[i] < tmpTemperatureMin THEN
				tmpTemperatureMin := gAMS.status.bank[j].resistorTemperature[i];
			END_IF;
		END_FOR;
		gAMS.data.bankResistorTemperatureMin[j] := tmpTemperatureMin;

	END_FOR;

	history;

END_PROGRAM

PROGRAM _EXIT
	(* Insert code here *)

END_PROGRAM
```

### Program Logical/AMS_and_Shunt/CAN/AMS_CAN/Receive
